// ---- FBs/Grid/FB_Grid_Power_Ext_Input.TcPOU
FUNCTION_BLOCK FB_Grid_Power_Ext_Input
VAR_INPUT PERSISTENT
	bEnable									: BOOL;													//Enable the Fuctionblock and his logic
	diNrOfEMS_IN							: DINT;													//Number of EMS on what this Device send Data
	rSizeGridConn							: REAL;													//{#lynus.ag#()} //Max Size of the Grid connection in kW
END_VAR
VAR_INPUT
	bExtErrorGrid							: BOOL;													//External Error for the Grid Function
	lrExtGridPower							: LREAL;												//External Grid power from a other Function or calculation in kW
	lrExtTotalCounterEnergy_Consumption		: LREAL;												//External Counter Value for Energy consumption with unit kWh
	lrExtTotalCounterEnergy_Production		: LREAL;												//External Counter Value for Energy production with unit kWh
	lrExtCounterEnergyT1_Consumption		: LREAL;												//External Counter Value for Energy consumption Tariff 1 with unit kWh
	lrExtCounterEnergyT2_Consumption		: LREAL;												//External Counter Value for Energy consumption Tariff 2 with unit kWh
	lrExtCounterEnergyT1_Production			: LREAL;												//External Counter Value for Energy production Tariff 1 with unit kWh
	lrExtCounterEnergyT2_Production			: LREAL;												//External Counter Value for Energy production Tariff 2 with unit kWh
END_VAR
VAR_OUTPUT
	stDataGrid								: ST_GridConnection_Output;								//{#lynus.ag#()} //Output Data from the Grid
	diNrOfGrid_OUT							: DINT;													//Active Number from the Grid connection for using on other functions
END_VAR
VAR
	{attribute 'hide'}
	fbGrid									: FB_GridConnection;									//Function block for grid connection
	{attribute 'hide'}
	fbNumberDevice							: FB_NumberOfDevice;									//Function block to calcualte the number of the Device
	{attribute 'hide'}
	timDissableFunctions					: TON;													//Timer to dissable the Function after Lynus_Standards.Constants_General.tTimeDissableLynusFunctions Days without connection to the Lynus Cloud
	{attribute 'hide'}
	timResetConnectionOnGVL					: TON;													//Timer to try reset the connection Flag on the GVL. (When somebody delete the Connection Function and make only a onlinechange)
	{attribute 'hide'}
	arrPD									: ARRAY[1..4] OF FB_PersistentData_Number;				//Function to save persistent data 
	{attribute 'hide'}
	byWaitInStep							: BYTE;													//Wait in Step before start to clean data on PLC
	{attribute 'hide'}
	iStateGVLData							: INT;													//State machine to handle the data on the GVL
	{attribute 'hide'}
	diCounterForGVL							: DINT;													//Counter to clean old data on GVL
	{attribute 'hide'}
	diLPForGVL								: DINT;													//Loop to clean old data on GVL
END_VAR
VAR PERSISTENT
	{attribute 'conditionalshow'}
	diNrOfEMS_IN_CP							: DINT;													//Number of EMS what control this Device to compare with the original
END_VAR

//Creator : Kai Ebensperger
//Company : Lynus AG
//Date : 07.06.2021
//Version : 1.0.0.0

//With this function block its possible to show the power data from a grid connection.
//The Power and Error Data came from a other Function and can connect to the Inputs. The Function write the Data then on the Lynus GVL
//The size from the Grid connection is sending to the ems

//NOTE for diNr.....Designation => 
//_IN = Here Data come in from other Functions or go out to other functions about the GVL
//_OUT = Here Data go out to other functions about the GVL

(*------------------------------------------------------------Limits----------------------------------------------------------------------------------*)

diNrOfEMS_IN := LIMIT(0,diNrOfEMS_IN,Constants_Energy.diMaxNumberOfEMS);

(*-------------------------------------------------------------Calcualte the number of Grid connection---------------------------------------------------------------*)

fbNumberDevice(
	diActualNumberOfDevices:= Lynus_Standards.GVL_Energy.stNumberOfDevices.diNumberOfGrids, 
	diMaxNumberOfDevices:= Constants_Energy.diMaxNumberOfGridConnections, 
	udiCounterOnlineChange:= TwinCAT_SystemInfoVarList._AppInfo.OnlineChangeCnt, 
	bNumberIsCalculatet=> , 
	bFPNumberIsCalculatet=> , 
	bOnlineChange=> , 
	diNumberForThisDevice=> diNrOfGrid_OUT, 
	diNumberOfTotalDevices=> );

//Write new Numer on GVL
IF fbNumberDevice.bFPNumberIsCalculatet THEN
	Lynus_Standards.GVL_Energy.stNumberOfDevices.diNumberOfGrids := fbNumberDevice.diNumberOfTotalDevices;	
END_IF 

//Delete old Number on GVL
IF fbNumberDevice.bOnlineChange THEN 
	Lynus_Standards.GVL_Energy.stNumberOfDevices.diNumberOfGrids := diNrOfGrid_OUT;	
		iStateGVLData := 1; 
END_IF	

(*-------------------------------------------------------------Service from Backend is ready and check the connection to backen for dissabel/enable Function---------------------------------------------------------------*)

//Try to reset the variable for connection on the GVL. When all is normal then the Lynus Mqtt connection function set this variable to true in the next cycle
//When we have no connection to the backend then after Lynus_Standards.Constants_General.tTimeDissableLynusFunctions days the Function is dissabled with all of his functionalities
timResetConnectionOnGVL(IN:= NOT timResetConnectionOnGVL.Q, PT:= T#1H, Q=> , ET=> );
	IF timResetConnectionOnGVL.Q THEN Lynus_Standards.GVL_Communicator.bStateConnectionToEnableFunctions := FALSE; END_IF
		IF NOT Lynus_Standards.GVL_Communicator.bStateConnectionToEnableFunctions THEN timDissableFunctions.IN := TRUE; ELSE timDissableFunctions.IN := FALSE; END_IF  
			timDissableFunctions(IN:= , PT:= Lynus_Standards.Constants_General.tTimeDissableLynusFunctions, Q=> , ET=> );

(*------------------------------------------------------------------Error----------------------------------------------------------------------------*)

IF timDissableFunctions.Q THEN fbGrid.bWarning := TRUE; fbGrid.iWarningCode := 0; ELSE fbGrid.bWarning := FALSE; END_IF 			
	IF bExtErrorGrid OR Lynus_Standards.GVL_Energy.stNumberOfDevices.diNumberOfGrids > Constants_Energy.diMaxNumberOfGridConnections THEN fbGrid.bError := TRUE; ELSE fbGrid.bError := FALSE; END_IF 

IF Lynus_Standards.GVL_Energy.stNumberOfDevices.diNumberOfGrids > Constants_Energy.diMaxNumberOfGridConnections THEN fbGrid.iErrorCode := 1;
ELSIF bExtErrorGrid THEN fbGrid.iErrorCode := 0;
END_IF  

(*------------------------------------------------------------------FB Grid----------------------------------------------------------------------------*)

fbGrid(
	bEnable:= bEnable AND NOT timDissableFunctions.Q, 
	bError:= , 
	bWriteWithDelay:= TRUE, 
	iErrorCode:= , 
	iWarningCode:= , 
	lrTotalCounterEnergy_Consumption:= lrExtTotalCounterEnergy_Consumption * 1000, 
	lrTotalCounterEnergy_Production:= lrExtTotalCounterEnergy_Production * 1000, 
	lrCounterEnergyT1_Consumption:= lrExtCounterEnergyT1_Consumption * 1000, 
	lrCounterEnergyT2_Consumption:= lrExtCounterEnergyT2_Consumption * 1000, 
	lrCounterEnergyT1_Production:= lrExtCounterEnergyT1_Production * 1000, 
	lrCounterEnergyT2_Production:= lrExtCounterEnergyT2_Production * 1000, 
	lrPowerGrid:= lrExtGridPower * 1000, 
	rSizeGridConn:= rSizeGridConn, 
	tTimDelayOutput:= T#5S, 
	stDataGridOut=> , 
	stDataGridOutDelay=> stDataGrid);
	
(*-----------------------------------------------------------Handle data to Global structure for the grid connections-----------------------------------------------------------------*)

//Delte al old Data on GVL after a online change or change on the variable diNrOfEMS_IDOD
IF diNrOfEMS_IN <> diNrOfEMS_IN_CP AND iStateGVLData = 0 THEN iStateGVLData := 10; END_IF 

CASE iStateGVLData OF
	
	0://Init Step
		byWaitInStep := 0;
			diCounterForGVL := 1;
	
	1://Wait for 4 Steps before clean al Data on GVL
		byWaitInStep := byWaitInStep + 1;
			IF byWaitInStep >= 4 AND fbNumberDevice.bNumberIsCalculatet THEN iStateGVLData := 2; END_IF
				//To much Devices, back to the Init step
				IF byWaitInStep >= 4 AND NOT fbNumberDevice.bNumberIsCalculatet THEN iStateGVLData := 0; END_IF	
			
	2://Clear all Data in GVL
		FOR diLPForGVL := 1 TO Constants_Energy.diMaxNumberOfEMS BY 1 DO 
			Lynus_Standards.GVL_Energy.stDataGridConnections[diLPForGVL,diCounterForGVL].bEnabled := FALSE;
				Lynus_Standards.GVL_Energy.stDataGridConnections[diLPForGVL,diCounterForGVL].byErrorWarning := 0;
					Lynus_Standards.GVL_Energy.stDataGridConnections[diLPForGVL,diCounterForGVL].lrPower := 0;
						Lynus_Standards.GVL_Energy.stDataGridConnections[diLPForGVL,diCounterForGVL].lrPowerConsumption := 0;
							Lynus_Standards.GVL_Energy.stDataGridConnections[diLPForGVL,diCounterForGVL].lrPowerProduction := 0;
								Lynus_Standards.GVL_Energy.stDataGridConnections[diLPForGVL,diCounterForGVL].rSizeGridConn := 0;
		END_FOR
			diCounterForGVL := diCounterForGVL + 1;
				diCounterForGVL := LIMIT(0,diCounterForGVL,Constants_Energy.diMaxNumberOfGridConnections);
					//Back to the init step
					IF diCounterForGVL >= Constants_Energy.diMaxNumberOfGridConnections THEN iStateGVLData := 0; END_IF

	10://Clear old Data on GVL 	
		Lynus_Standards.GVL_Energy.stDataGridConnections[diNrOfEMS_IN_CP,diNrOfGrid_OUT].bEnabled := FALSE;
			Lynus_Standards.GVL_Energy.stDataGridConnections[diNrOfEMS_IN_CP,diNrOfGrid_OUT].byErrorWarning := 0;
				Lynus_Standards.GVL_Energy.stDataGridConnections[diNrOfEMS_IN_CP,diNrOfGrid_OUT].lrPower := 0;
					Lynus_Standards.GVL_Energy.stDataGridConnections[diNrOfEMS_IN_CP,diNrOfGrid_OUT].lrPowerConsumption := 0;
						Lynus_Standards.GVL_Energy.stDataGridConnections[diNrOfEMS_IN_CP,diNrOfGrid_OUT].lrPowerProduction := 0;
							Lynus_Standards.GVL_Energy.stDataGridConnections[diNrOfEMS_IN_CP,diNrOfGrid_OUT].rSizeGridConn := 0;
	
		diNrOfEMS_IN_CP := diNrOfEMS_IN;
			//Back to the init step
			iStateGVLData := 0;

END_CASE 	 

IF diNrOfGrid_OUT > 0 AND fbNumberDevice.bNumberIsCalculatet AND diNrOfEMS_IN > 0 THEN
	Lynus_Standards.GVL_Energy.stDataGridConnections[diNrOfEMS_IN,diNrOfGrid_OUT].bEnabled := fbGrid.stDataGridOut.bEnabled;
		Lynus_Standards.GVL_Energy.stDataGridConnections[diNrOfEMS_IN,diNrOfGrid_OUT].byErrorWarning := fbGrid.stDataGridOut.byErrorWarning;
			Lynus_Standards.GVL_Energy.stDataGridConnections[diNrOfEMS_IN,diNrOfGrid_OUT].lrPower := fbGrid.stDataGridOut.lrPower;
				Lynus_Standards.GVL_Energy.stDataGridConnections[diNrOfEMS_IN,diNrOfGrid_OUT].lrPowerConsumption := fbGrid.stDataGridOut.lrPowerConsumption;
					Lynus_Standards.GVL_Energy.stDataGridConnections[diNrOfEMS_IN,diNrOfGrid_OUT].lrPowerProduction := fbGrid.stDataGridOut.lrPowerProduction;
						Lynus_Standards.GVL_Energy.stDataGridConnections[diNrOfEMS_IN,diNrOfGrid_OUT].rSizeGridConn := fbGrid.stDataGridOut.rSizeGridConn;
END_IF

(*----------------------------------------------------------Save persistent data----------------------------------------------------------------*)

arrPD[1](lrValue:= BOOL_TO_LREAL(bEnable), bEventBasedActive=> );
arrPD[2](lrValue:= DINT_TO_LREAL(diNrOfEMS_IN), bEventBasedActive=> );
arrPD[3](lrValue:= REAL_TO_LREAL(rSizeGridConn), bEventBasedActive=> );
arrPD[4](lrValue:= DINT_TO_LREAL(diNrOfEMS_IN_CP), bEventBasedActive=> );

END_FUNCTION_BLOCK

// ---- FBs/KBus State/FB_K_Bus_State_old.TcPOU
FUNCTION_BLOCK FB_K_Bus_State_old
VAR_INPUT
END_VAR
VAR_OUTPUT
	uiKBusState_OUT					AT%I*		: UINT;											//K-Bus State from the Basestation on wich the Terminal KL6301 is connected
END_VAR
VAR
END_VAR

//Creator : Kai Ebensperger
//Company : Lynus AG
//Date : 24.07.2021
//Version : 1.0.0.0

//With this Function Block its possible to connect the Variable on the output to the State Variable with the K-Bus Box
//In this Function we dont need code

END_FUNCTION_BLOCK

// ---- FBs/KBus State/FB_K_Bus_State.TcPOU
FUNCTION_BLOCK FB_K_Bus_State
VAR_INPUT
END_VAR
VAR_OUTPUT
	uiKBusState_OUT					AT%I*		: UINT;											//K-Bus State from the Basestation on wich the Terminal KL6301 is connected
	b_Kbus_notOk			: BOOL;			// KBus not OK, State <> 0
	word_ErrorCount			: WORD;			// Counts 1 up every time the KBus gets reset
END_VAR
VAR
	FB_IOF_DeviceReset	: IOF_DeviceReset;
    DEVICEID  : UDINT;
    RESET     : BOOL;
	ton_Delay_ResetKBus: Ton;
	Count_up: CTU;
END_VAR

//Creator : Stefan Lackner
//Company : EfficientIO
//Date : 09.02.2023
//Version : 1.0.0.0

//With this Function Block its possible to connect the Variable on the output to the State Variable with the K-Bus Box
//if the State <> 0 for longer then one Minute, the KBus gets reset

IF uiKBusState_OUT <> 0 AND NOT FB_IOF_DeviceReset.BUSY THEN
	ton_Delay_ResetKBus.IN := TRUE;
ELSE
	ton_Delay_ResetKBus.IN := FALSE;
END_IF
ton_Delay_ResetKBus( PT := T#1M);
 
FB_IOF_DeviceReset(
	NETID:= '', 
	DEVICEID:= 2, 		// ID 2 is the first terminal
	RESET:= ton_Delay_ResetKBus.Q, 
	TMOUT:= T#5S, 
	BUSY=> , 
	ERR=> , 
	ERRID=> );
	
IF uiKBusState_OUT <> 0 THEN
	b_Kbus_notOk := TRUE;
ELSE
	b_Kbus_notOk := FALSE;
END_IF

Count_up(
	CU:= b_Kbus_notOk, 
	RESET:= FALSE , 
	PV:= , 
	Q=> , 
	CV=> word_ErrorCount);

END_FUNCTION_BLOCK

// ---- FBs/MBus Master/FB_KL6781_MBus_Master.TcPOU
FUNCTION_BLOCK FB_KL6781_MBus_Master
VAR_INPUT PERSISTENT
	eBaudrateMBus							: E_MBus_Baudrate;				//With this Baudrate the Functionsblocks for the Counters are reading out
END_VAR
VAR_OUTPUT
	bBusy									: BOOL;							//Function is Busy
	bReady									: BOOL;							//Function is Ready
	byErrorWarning							: BYTE;							//Error Warning State
	diNrOfMBusMasterLine_OUT				: DINT;							//Active Number from the MBus Master Function for using on other functions
	eMessageMBusMaster						: E_Message_MBusMaster;			//Message from the MBus Master Function
END_VAR
VAR
	{attribute 'hide'}
	fbMbusMaster							: FB_MBUSKL6781;				//MBus Master for KL6781
	{attribute 'hide'}
	fbNumberDevice							: FB_NumberOfDevice;			//Function block to calcualte the number of the Device
	{attribute 'hide'}
	fbMBusMessage							: FB_MBusMaster_Messages;		//MBus Messages
	{attribute 'hide'}
	fbPD									: FB_PersistentData_Number;		//FB Persistent Data
	{attribute 'hide'}
	timDissableFunctions					: TON;							//Timer to dissable the Function after Lynus_Standards.Constants_General.tTimeDissableLynusFunctions Days without connection to the Lynus Cloud
	{attribute 'hide'}
	timResetConnectionOnGVL					: TON;							//Timer to try reset the connection Flag on the GVL. (When somebody delete the Connection Function and make only a onlinechange)
	stMBusKL6781ComIn        	AT%I*	 	: ST_KL6781inData22B;			//Input Structure for the KL6781 to map on the KL6781 Terminal
	stMBusKL6781ComOut        	AT%Q*		: ST_KL6781outData22B;			//Output Structure for the KL6781 to map on the KL6781 Terminal
	{attribute 'hide'}
	byWaitInStep							: BYTE;							//Wait in Step before start to clean data on PLC
	{attribute 'hide'}
	iStateGVLData							: INT;							//State machine to handle the data on the GVL
	{attribute 'hide'}
	diCounterForGVL							: DINT;							//Counter to clean old data on GVL
END_VAR

//Creator : Kai Ebensperger
//Company : Lynus AG
//Date : 23.07.2021
//Version : 1.0.0.0

//With this function block we can communicate with a beckhoff KL6781 MBus Terminal.
//This Functionblock receive the requests from the other Counter Functions and send to the Hardware Counters in the field.
//The answer from the Hardware Counters comes back to this Function and then they distribute to the Counter Function in the plc.
//This Function must be called in a task of < 10MS. Is depends about the Baudrate. 2400Baud = 10MS Task
//The request to a Hardware counter and the response is min. 1 second on MBus.


//NOTE for diNr.....Designation => 
//_IN = Here Data come in from other Functions or go out to other functions about the GVL
//_OUT = Here Data go out to other functions about the GVL

(*-------------------------------------------------------------Calcualte the number of MBus Master---------------------------------------------------------------*)

fbNumberDevice(
	diActualNumberOfDevices:= Lynus_Standards.GVL_Bussystems.diNumberOfMBusMasters, 
	diMaxNumberOfDevices:= Constants_Bussystems.diMaxNumberOfMBusMasterKL6781, 
	udiCounterOnlineChange:= TwinCAT_SystemInfoVarList._AppInfo.OnlineChangeCnt, 
	bNumberIsCalculatet=> , 
	bFPNumberIsCalculatet=> , 
	bOnlineChange=> , 
	diNumberForThisDevice=> diNrOfMBusMasterLine_OUT, 
	diNumberOfTotalDevices=> );

//Write new Numer on GVL
IF fbNumberDevice.bFPNumberIsCalculatet THEN
	Lynus_Standards.GVL_Bussystems.diNumberOfMBusMasters := fbNumberDevice.diNumberOfTotalDevices;	
END_IF 

//Delete old Number on GVL
IF fbNumberDevice.bOnlineChange THEN 
	Lynus_Standards.GVL_Bussystems.diNumberOfMBusMasters := diNrOfMBusMasterLine_OUT;	
		iStateGVLData := 1; 
END_IF	

(*-------------------------------------------------------------Service from Backend is ready and check the connection to backen for dissabel/enable Function---------------------------------------------------------------*)

//Try to reset the variable for connection on the GVL. When all is normal then the Lynus Mqtt connection function set this variable to true in the next cycle
//When we have no connection to the backend then after Lynus_Standards.Constants_General.tTimeDissableLynusFunctions days the Function is dissabled with all of his functionalities
timResetConnectionOnGVL(IN:= NOT timResetConnectionOnGVL.Q, PT:= T#1H, Q=> , ET=> );
	IF timResetConnectionOnGVL.Q THEN Lynus_Standards.GVL_Communicator.bStateConnectionToEnableFunctions := FALSE; END_IF
		IF NOT Lynus_Standards.GVL_Communicator.bStateConnectionToEnableFunctions THEN timDissableFunctions.IN := TRUE; ELSE timDissableFunctions.IN := FALSE; END_IF  
			timDissableFunctions(IN:= , PT:= Lynus_Standards.Constants_General.tTimeDissableLynusFunctions, Q=> , ET=> );
			
(*-------------------------------------------------------------M-Bus Master---------------------------------------------------------------*)

fbMbusMaster(
	usiRetries:= 0, 
	bStart:= , 
	bDisabled:= timDissableFunctions.Q OR diNrOfMBusMasterLine_OUT <= 0 OR NOT fbNumberDevice.bNumberIsCalculatet , 
	bBusy=> bBusy, 
	bReady=> bReady, 
	bError=> , 
	eError=> , 
	stComIn:= stMBusKL6781ComIn, 
	stComOut:= stMBusKL6781ComOut, 
	stCom:= Lynus_Standards.GVL_Bussystems.stDataOfMBusMasterKL6781[diNrOfMBusMasterLine_OUT].stDataMBusCommunicationKL6781);
	
(*------------------------------------------------------------------Error and Warning----------------------------------------------------------------------------*)
			
IF timDissableFunctions.Q THEN fbMBusMessage.bWarning := TRUE; fbMBusMessage.iWarningCode := 0; ELSE fbMBusMessage.bWarning := FALSE; END_IF   
	IF (Lynus_Standards.GVL_Bussystems.diNumberOfMBusMasters > Constants_Bussystems.diMaxNumberOfMBusMasterKL6781) THEN 
		fbMBusMessage.bErrorIntern := TRUE;
			fbMBusMessage.iErrorCode := 1;
	ELSE
		fbMBusMessage.bErrorIntern := FALSE;
	END_IF	

IF fbMbusMaster.bError THEN 
	fbMBusMessage.bErrorMBus := TRUE;
		fbMBusMessage.iErrorCode := fbMbusMaster.eError;
ELSE
	IF NOT fbMbusMaster.bError AND NOT fbMbusMaster.bBusy THEN 
		fbMBusMessage.bErrorMBus := FALSE;
	END_IF
END_IF	
		
fbMBusMessage(
	bErrorMBus:= , 
	bErrorIntern:= , 
	bWarning:= , 
	iWarningCode:= , 
	iErrorCode:= , 
	byErrorWarning=> byErrorWarning, 
	eMessageMBusMaster=> eMessageMBusMaster);
	
(*-----------------------------------------------------------Handle data to Global structure for MBus Communication-----------------------------------------------------------------*)
	
CASE iStateGVLData OF
	
	0://Init Step
		byWaitInStep := 0;
			diCounterForGVL := 1;
	
	1://Wait for 4 Steps before clean al Data on GVL
		byWaitInStep := byWaitInStep + 1;
			IF byWaitInStep >= 4 AND fbNumberDevice.bNumberIsCalculatet THEN iStateGVLData := 2; END_IF
				//To much Devices, back to the Init step
				IF byWaitInStep >= 4 AND NOT fbNumberDevice.bNumberIsCalculatet THEN iStateGVLData := 0; END_IF	
			
	2://Clear all Data in GVL
	//Some Parts in the GVL Reset the Slave. Otherwise there will be problems when writing the new addresses to the array in the GVL.
	
		Lynus_Standards.GVL_Bussystems.stDataOfMBusMasterKL6781[diCounterForGVL].eBaudrateMBusKL6781 := E_MBus_Baudrate.eMBus_NoBaudrate;
														 		
		diCounterForGVL := diCounterForGVL + 1;
			diCounterForGVL := LIMIT(0,diCounterForGVL,Constants_Bussystems.diMaxNumberOfMBusMasterKL6781);
				//Back to the init step
				IF diCounterForGVL >= Constants_Bussystems.diMaxNumberOfMBusMasterKL6781 THEN iStateGVLData := 0; END_IF

END_CASE 
	
IF diNrOfMBusMasterLine_OUT > 0 AND fbNumberDevice.bNumberIsCalculatet THEN  
	Lynus_Standards.GVL_Bussystems.stDataOfMBusMasterKL6781[diNrOfMBusMasterLine_OUT].eBaudrateMBusKL6781 := eBaudrateMBus;
END_IF	

(*----------------------------------------------------------Save persistent data----------------------------------------------------------------*)

fbPD(lrValue:= INT_TO_LREAL(eBaudrateMBus), bEventBasedActive=> );

END_FUNCTION_BLOCK

// ---- FBs/Meter/Beckhoff/Electric KL3403/FB_EM_Beckhoff_KL3403.TcPOU
FUNCTION_BLOCK FB_EM_Beckhoff_KL3403
VAR_INPUT PERSISTENT
	bEnable							: BOOL;											//Enable the function
	bChannel1Invers					: BOOL;											//Invert the Output data from Channel 1. = L1
	bChannel2Invers					: BOOL;											//Invert the Output data from Channel 2. = L2
	bChannel3Invers					: BOOL;											//Invert the Output data from Channel 3. = L3
	uiCurrentTransformerRatioL1		: UINT;											//Current Transformer Ratio for Channel 1 (L1)
	uiCurrentTransformerRatioL2		: UINT;											//Current Transformer Ratio for Channel 2 (L2)
	uiCurrentTransformerRatioL3		: UINT;											//Current Transformer Ratio for Channel 3 (L3)
END_VAR
VAR_INPUT
	uiKBusState_IN					: UINT;											//K-Bus State from the K-Bus Box on wich the Terminal is connected. (Connect with FB_K_Bus_state)
END_VAR
VAR_OUTPUT
	stDataEMPower					: ST_ElectricMeter_Output_Power;				//Output structure with Data from Electric Meter (Power Data)
	stDataEMCounter					: ST_ElectricMeter_Output_Counter;				//Output structure with Data from Electric Meter (Counter Data)
	stDataEMPowerRealTime			: ST_ElectricMeter_Output_Power;				//Output structure with Data from Electric Meter (Power Data RealTime)
	stDataEMCounterRealTime			: ST_ElectricMeter_Output_Counter;				//Output structure with Data from Electric Meter (Counter Data RealTime)
	diNrOfEM_OUT					: DINT;											//Active Number from the Electric Meter for using on other functions
END_VAR
VAR
	{attribute 'conditionalshow'}
	fbEM							: FB_ElectricMeter;								//Electric Meter Function
	{attribute 'conditionalshow'}
	fbEnergyCounter					: FB_EnergyCounter;								//FB energy Counter, because the KL3403 has no nice logic for the Energy value
	{attribute 'hide'}
	fbNumberDevice					: FB_NumberOfDevice;							//Function block to calcualte the number of the Device
	fbKL3403						: FB_KL3403_SimpleProcessImage;					//Function KL3403
	{attribute 'hide'}
	stDataL1						: ST_KL3403;									//Data from Channel 1 (L1)
	{attribute 'hide'}
	stDataL2						: ST_KL3403;									//Data from Channel 2 (L2)
	{attribute 'hide'}
	stDataL3						: ST_KL3403;									//Data from Channel 3 (L3)
	{attribute 'hide'}
	timDissableFunctions			: TON;											//Timer to dissable the Function after Lynus_Standards.Constants_General.tTimeDissableLynusFunctions Days without connection to the Lynus Cloud
	{attribute 'hide'}
	timResetConnectionOnGVL			: TON;											//Timer to try reset the connection Flag on the GVL. (When somebody delete the Connection Function and make only a onlinechange)
	{attribute 'hide'}
	timSetCounterValues				: TON;											//Timer to set the counter values from the KL3403 Function to the EM Function
	{attribute 'hide'}
	arrPD							: ARRAY[1..7] OF FB_PersistentData_Number;		//Function to save persistent data
	{attribute 'hide'}
	byWaitInStep					: BYTE;											//Wait in Step before start to clean data on PLC
	{attribute 'hide'}
	iStateGVLData					: INT;											//State machine to handle the data on the GVL
	{attribute 'hide'}
	diCounterForGVL					: DINT;											//Counter to clean old data on GVL
END_VAR

//Creator : Kai Ebensperger
//Company : Lynus AG
//Date : 04.10.2021
//Version : 1.0.0.0

//Stefan: Addes S and Q calculation

//With this function is possible to read out all Information from a KL3403
//This Function support only the Simple Process Image and the Ratio in the Terminal register must be Set allways to 1.

//NOTE for diNr.....Designation => 
//_IN = Here Data come in from other Functions or go out to other functions about the GVL
//_OUT = Here Data go out to other functions about the GVL

(*-------------------------------------------------------------Calcualte the number of EM---------------------------------------------------------------*)

fbNumberDevice(
	diActualNumberOfDevices:= Lynus_Standards.GVL_Energy.stNumberOfDevices.diNumberOfElectricMeters, 
	diMaxNumberOfDevices:= Constants_Energy.diMaxNumberOfElectricMeters, 
	udiCounterOnlineChange:= TwinCAT_SystemInfoVarList._AppInfo.OnlineChangeCnt, 
	bNumberIsCalculatet=> , 
	bFPNumberIsCalculatet=> , 
	bOnlineChange=> , 
	diNumberForThisDevice=> diNrOfEM_OUT, 
	diNumberOfTotalDevices=> );

//Write new Numer on GVL
IF fbNumberDevice.bFPNumberIsCalculatet THEN
	Lynus_Standards.GVL_Energy.stNumberOfDevices.diNumberOfElectricMeters := fbNumberDevice.diNumberOfTotalDevices;	
END_IF

//Delete old Number on GVL
IF fbNumberDevice.bOnlineChange THEN 
	Lynus_Standards.GVL_Energy.stNumberOfDevices.diNumberOfElectricMeters := diNrOfEM_OUT;	
		iStateGVLData := 1; 
END_IF

(*-------------------------------------------------------------Service from Backend is ready and check the connection to backen for dissabel/enable Function---------------------------------------------------------------*)

//Try to reset the variable for connection on the GVL. When all is normal then the Lynus Mqtt connection function set this variable to true in the next cycle
//When we have no connection to the backend then after Lynus_Standards.Constants_General.tTimeDissableLynusFunctions days the Function is dissabled with all of his functionalities
timResetConnectionOnGVL(IN:= NOT timResetConnectionOnGVL.Q, PT:= T#1H, Q=> , ET=> );
	IF timResetConnectionOnGVL.Q THEN Lynus_Standards.GVL_Communicator.bStateConnectionToEnableFunctions := FALSE; END_IF
		IF NOT Lynus_Standards.GVL_Communicator.bStateConnectionToEnableFunctions THEN timDissableFunctions.IN := TRUE; ELSE timDissableFunctions.IN := FALSE; END_IF  
			timDissableFunctions(IN:= , PT:= Lynus_Standards.Constants_General.tTimeDissableLynusFunctions, Q=> , ET=> );

(*----------------------------------------------------------------------------------------KL3403 Communication----------------------------------------------------------------------------------------------*)

fbKL3403(
	uiKBusState_IN:= uiKBusState_IN, 
	uiCurrentTransformerRatioL1:= uiCurrentTransformerRatioL1,
	uiCurrentTransformerRatioL2:= uiCurrentTransformerRatioL2,
	uiCurrentTransformerRatioL3:= uiCurrentTransformerRatioL3,
	rResolutionCurrent:= 0.001,
	rResolutionPower:= 0.1,
	rResolutionEnergy:= 0.01,
	stDataL1=> , 
	stDataL2=> ,
	stDataL3=> );

//Invert the Output data, because it is possible that the current transformers have been mounted in different mounting positions.
IF NOT bChannel1Invers THEN
	stDataL1 := fbKL3403.stDataL1;
ELSE
	stDataL1.byErrorWarning := fbKL3403.stDataL1.byErrorWarning;
	stDataL1.rCurrent := fbKL3403.stDataL1.rCurrent;
	stDataL1.rVoltage := fbKL3403.stDataL1.rVoltage;
	stDataL1.rPower := fbKL3403.stDataL1.rPower * - 1;
	stDataL1.rPowerfactor := fbKL3403.stDataL1.rPowerfactor;
	stDataL1.rEnergy := fbKL3403.stDataL1.rEnergy;
	stDataL1.rFrequency := fbKL3403.stDataL1.rFrequency;
	stDataL1.rPeakValueCurrent := fbKL3403.stDataL1.rPeakValueCurrent;
	stDataL1.rPeakValueVoltage := fbKL3403.stDataL1.rPeakValueVoltage;
	stDataL1.rPeakValuePower := fbKL3403.stDataL1.rPeakValuePower * - 1;
	stDataL1.rMinValueCurrent := fbKL3403.stDataL1.rMinValueCurrent;
	stDataL1.rMinValueVoltage := fbKL3403.stDataL1.rMinValueVoltage;
	stDataL1.rMinValuePower := fbKL3403.stDataL1.rMinValuePower * - 1;
END_IF

IF NOT bChannel2Invers THEN
	stDataL2 := fbKL3403.stDataL2;
ELSE
	stDataL2.byErrorWarning := fbKL3403.stDataL2.byErrorWarning;
	stDataL2.rCurrent := fbKL3403.stDataL2.rCurrent;
	stDataL2.rVoltage := fbKL3403.stDataL2.rVoltage;
	stDataL2.rPower := fbKL3403.stDataL2.rPower * - 1;
	stDataL2.rPowerfactor := fbKL3403.stDataL2.rPowerfactor;
	stDataL2.rEnergy := fbKL3403.stDataL2.rEnergy;
	stDataL2.rFrequency := fbKL3403.stDataL2.rFrequency;
	stDataL2.rPeakValueCurrent := fbKL3403.stDataL2.rPeakValueCurrent;
	stDataL2.rPeakValueVoltage := fbKL3403.stDataL2.rPeakValueVoltage;
	stDataL2.rPeakValuePower := fbKL3403.stDataL2.rPeakValuePower * - 1;
	stDataL2.rMinValueCurrent := fbKL3403.stDataL2.rMinValueCurrent;
	stDataL2.rMinValueVoltage := fbKL3403.stDataL2.rMinValueVoltage;
	stDataL2.rMinValuePower := fbKL3403.stDataL2.rMinValuePower * - 1;
END_IF

IF NOT bChannel3Invers THEN
	stDataL3 := fbKL3403.stDataL3;
ELSE
	stDataL3.byErrorWarning := fbKL3403.stDataL3.byErrorWarning;
	stDataL3.rCurrent := fbKL3403.stDataL3.rCurrent;
	stDataL3.rVoltage := fbKL3403.stDataL3.rVoltage;
	stDataL3.rPower := fbKL3403.stDataL3.rPower * - 1;
	stDataL3.rPowerfactor := fbKL3403.stDataL3.rPowerfactor;
	stDataL3.rEnergy := fbKL3403.stDataL3.rEnergy;
	stDataL3.rFrequency := fbKL3403.stDataL3.rFrequency;
	stDataL3.rPeakValueCurrent := fbKL3403.stDataL3.rPeakValueCurrent;
	stDataL3.rPeakValueVoltage := fbKL3403.stDataL3.rPeakValueVoltage;
	stDataL3.rPeakValuePower := fbKL3403.stDataL3.rPeakValuePower * - 1;
	stDataL3.rMinValueCurrent := fbKL3403.stDataL3.rMinValueCurrent;
	stDataL3.rMinValueVoltage := fbKL3403.stDataL3.rMinValueVoltage;
	stDataL3.rMinValuePower := fbKL3403.stDataL3.rMinValuePower * - 1;
END_IF
	
(*----------------------------------------------------------------------------------------Energy Counter Function----------------------------------------------------------------------------------------------*)

//For the KL3403 we use a external Energy Counter Function. So we can count Import and Export Energy with the KL3403.
//Attetntion, the KL3403 is not MID Conform. Thus, these values must not be used for billing.
fbEnergyCounter(
	byActiveTariff:= 1, 
	lrPowerInput:= (stDataL1.rPower + stDataL2.rPower + stDataL3.rPower) / 1000, 
	lrTotalCounterEnergy_Consumption=> , 
	lrTotalCounterEnergy_Production=> , 
	lrCounterEnergyT1_Consumption=> , 
	lrCounterEnergyT2_Consumption=> , 
	lrCounterEnergyT1_Production=> , 
	lrCounterEnergyT2_Production=> );

(*----------------------------------------------------------------------------------------Electric Meter Function----------------------------------------------------------------------------------------------*)

//Error
IF timDissableFunctions.Q THEN fbEM.bWarning := TRUE; fbEM.iWarningCode := 0; ELSE fbEM.bWarning := FALSE; END_IF 
	IF Lynus_Standards.GVL_Energy.stNumberOfDevices.diNumberOfElectricMeters > Constants_Energy.diMaxNumberOfElectricMeters OR 
		stDataL1.byErrorWarning = 2 OR stDataL2.byErrorWarning = 2 OR stDataL3.byErrorWarning = 2 THEN 
			fbEM.bError := TRUE; 
	ELSE 
			fbEM.bError := FALSE; 
	END_IF
		IF Lynus_Standards.GVL_Energy.stNumberOfDevices.diNumberOfElectricMeters > Constants_Energy.diMaxNumberOfElectricMeters THEN fbEM.iErrorCode := 1;
		ELSIF stDataL1.byErrorWarning = 2 OR stDataL2.byErrorWarning = 2 OR stDataL3.byErrorWarning = 2 THEN fbEM.iErrorCode := 0;
		END_IF

timSetCounterValues(IN:= bEnable AND NOT timSetCounterValues.Q, PT:= T#2S, Q=> , ET=> );		

//Function
fbEM(
	bEnable:= bEnable AND NOT timDissableFunctions.Q, 
	bError:= , 
	bEnableReadOutFunction:= FALSE, 
	bWriteWithDelay:= TRUE, 
	bPowerDataInvers:= FALSE,
	bReadOutDataDone:= timSetCounterValues.Q,
	iTimeReadOutInterval:= 0, 
	iErrorCode:= , 
	iWarningCode:= , 
	lrTotalCounterEnergy_Consumption:= fbEnergyCounter.lrTotalCounterEnergy_Consumption,
	lrTotalCounterEnergy_Production:= fbEnergyCounter.lrTotalCounterEnergy_Production, 
	lrCounterEnergyT1_Consumption:= fbEnergyCounter.lrCounterEnergyT1_Consumption,
	lrCounterEnergyT2_Consumption:= fbEnergyCounter.lrCounterEnergyT2_Consumption,
	lrCounterEnergyT1_Production:= fbEnergyCounter.lrCounterEnergyT1_Production, 
	lrCounterEnergyT2_Production:= fbEnergyCounter.lrCounterEnergyT2_Production, 
	lrCurrentL1:= stDataL1.rCurrent, 
	lrVoltageL1N:= stDataL1.rVoltage, 
	lrVoltageL1L2:= stDataL1.rVoltage*SQRT(3), 
	lrPowerL1:= stDataL1.rPower, 
	lrCurrentL2:= stDataL2.rCurrent, 
	lrVoltageL2N:= stDataL2.rVoltage, 
	lrVoltageL2L3:= stDataL2.rVoltage*SQRT(3), 
	lrPowerL2:= stDataL2.rPower, 
	lrCurrentL3:= stDataL3.rCurrent, 
	lrVoltageL3N:= stDataL3.rVoltage, 
	lrVoltageL3L1:= stDataL3.rVoltage*SQRT(3), 
	lrPowerL3:= stDataL3.rPower, 
	lrPowerTotal:= stDataL1.rPower + stDataL2.rPower + stDataL3.rPower, 
	lrFrequency:= (stDataL1.rFrequency + stDataL2.rFrequency + stDataL3.rFrequency) / 3, 
 	lrApparentPowerTotal:=,
	lrReactivePowerTotal:=, 
	tTimDelayOutput:= T#5S, 
	stDataEMOutPower=> stDataEMPowerRealTime, 
	stDataEMOutPowerDelay=> stDataEMPower, 
	stDataEMOutCounter=> stDataEMCounterRealTime,
	stDataEMOutCounterDelay=> stDataEMCounter,
	bReadOutMeter=> );
(*
	IF  stDataL1.rPowerfactor <>0 AND stDataL2.rPowerfactor <>0 AND stDataL3.rPowerfactor <>0 THEN
		fbEM.lrApparentPowerTotal:= ABS(stDataL1.rPower)/ABS(stDataL1.rPowerfactor) + ABS(stDataL2.rPower)/ABS(stDataL2.rPowerfactor) + ABS(stDataL3.rPower)/ABS(stDataL3.rPowerfactor); 
	END_IF	
*)


	//calculate total apparant power in VA
	fbEM.lrApparentPowerTotal := fbEM.lrVoltageL1N * fbEM.lrCurrentL1 + fbEM.lrVoltageL2N * fbEM.lrCurrentL2 +  fbEM.lrVoltageL3N * fbEM.lrCurrentL3;
	
	IF fbEM.lrApparentPowerTotal<>0 AND fbEM.lrPowerTotal<>0 AND fbEM.lrApparentPowerTotal> ABS(fbEM.lrPowerTotal) THEN
		fbEM.lrReactivePowerTotal:= SQRT(ABS(fbEM.lrApparentPowerTotal*fbEM.lrApparentPowerTotal - ABS(fbEM.lrPowerTotal*fbEM.lrPowerTotal)));	
	END_IF
	IF stDataL1.rPowerfactor<>0 AND stDataL2.rPowerfactor <>0 AND stDataL3.rPowerfactor<>0 THEN 	// check that not all cos phi are not 0
		IF (stDataL1.rPowerfactor+stDataL2.rPowerfactor+stDataL3.rPowerfactor)<>0 THEN				// check that the sum is not 0	
			IF 	(stDataL1.rPowerfactor+stDataL2.rPowerfactor+stDataL3.rPowerfactor)/3<0 THEN		// check is the average is below 0 / capacitive
				fbEM.lrReactivePowerTotal:=fbEM.lrReactivePowerTotal*(-1);
			END_IF
		END_IF	
	END_IF
(*-----------------------------------------------------------Handle data to Global structure for Electric Meter-----------------------------------------------------------------*)

CASE iStateGVLData OF
	
	0://Init Step
		byWaitInStep := 0;
			diCounterForGVL := 1;
	
	1://Wait for 4 Steps before clean al Data on GVL
		byWaitInStep := byWaitInStep + 1;
			IF byWaitInStep >= 4 AND fbNumberDevice.bNumberIsCalculatet THEN iStateGVLData := 2; END_IF
				//To much Devices, back to the Init step
				IF byWaitInStep >= 4 AND NOT fbNumberDevice.bNumberIsCalculatet THEN iStateGVLData := 0; END_IF	
			
	2://Clear all Data in GVL
		Lynus_Standards.GVL_Energy.stDataElectricMeters[diCounterForGVL].bEnabled := FALSE;	
			Lynus_Standards.GVL_Energy.stDataElectricMeters[diCounterForGVL].byErrorWarning := 0;
				Lynus_Standards.GVL_Energy.stDataElectricMeters[diCounterForGVL].lrCounterEnergyT1_Consumption := 0;
					Lynus_Standards.GVL_Energy.stDataElectricMeters[diCounterForGVL].lrCounterEnergyT1_Production := 0;
						Lynus_Standards.GVL_Energy.stDataElectricMeters[diCounterForGVL].lrCounterEnergyT2_Consumption := 0;
							Lynus_Standards.GVL_Energy.stDataElectricMeters[diCounterForGVL].lrCounterEnergyT2_Production := 0;
								Lynus_Standards.GVL_Energy.stDataElectricMeters[diCounterForGVL].lrPower := 0;
									Lynus_Standards.GVL_Energy.stDataElectricMeters[diCounterForGVL].lrPowerConsumption := 0;
										Lynus_Standards.GVL_Energy.stDataElectricMeters[diCounterForGVL].lrPowerProduction := 0;
											Lynus_Standards.GVL_Energy.stDataElectricMeters[diCounterForGVL].lrTotalCounterEnergy_Consumption := 0;
												Lynus_Standards.GVL_Energy.stDataElectricMeters[diCounterForGVL].lrTotalCounterEnergy_Production := 0;
		
		//Electric Meters
		diCounterForGVL := diCounterForGVL + 1;
			diCounterForGVL := LIMIT(0,diCounterForGVL,Constants_Energy.diMaxNumberOfElectricMeters);
				//Back to the init step
				IF diCounterForGVL >= Constants_Energy.diMaxNumberOfElectricMeters THEN iStateGVLData := 0; END_IF

END_CASE 	 

//Write Data on GVL for Electric Meter
IF diNrOfEM_OUT > 0 AND fbNumberDevice.bNumberIsCalculatet THEN
	Lynus_Standards.GVL_Energy.stDataElectricMeters[diNrOfEM_OUT].bEnabled := fbEM.stDataEMOutPower.bEnabled;
		Lynus_Standards.GVL_Energy.stDataElectricMeters[diNrOfEM_OUT].byErrorWarning := fbEM.stDataEMOutPower.byErrorWarning;
			Lynus_Standards.GVL_Energy.stDataElectricMeters[diNrOfEM_OUT].lrCounterEnergyT1_Consumption := fbEM.stDataEMOutCounter.lrCounterEnergyT1_Consumption;
				Lynus_Standards.GVL_Energy.stDataElectricMeters[diNrOfEM_OUT].lrCounterEnergyT1_Production := fbEM.stDataEMOutCounter.lrCounterEnergyT1_Production;
					Lynus_Standards.GVL_Energy.stDataElectricMeters[diNrOfEM_OUT].lrCounterEnergyT2_Consumption := fbEM.stDataEMOutCounter.lrCounterEnergyT2_Consumption;
						Lynus_Standards.GVL_Energy.stDataElectricMeters[diNrOfEM_OUT].lrCounterEnergyT2_Production := fbEM.stDataEMOutCounter.lrCounterEnergyT2_Production;		
							Lynus_Standards.GVL_Energy.stDataElectricMeters[diNrOfEM_OUT].lrPower := fbEM.stDataEMOutPower.lrPowerTotal;
								Lynus_Standards.GVL_Energy.stDataElectricMeters[diNrOfEM_OUT].lrPowerConsumption := fbEM.stDataEMOutPower.lrPowerConsumption;
									Lynus_Standards.GVL_Energy.stDataElectricMeters[diNrOfEM_OUT].lrPowerProduction := fbEM.stDataEMOutPower.lrPowerProduction;
										Lynus_Standards.GVL_Energy.stDataElectricMeters[diNrOfEM_OUT].lrTotalCounterEnergy_Consumption := fbEM.stDataEMOutCounter.lrTotalCounterEnergy_Consumption;
											Lynus_Standards.GVL_Energy.stDataElectricMeters[diNrOfEM_OUT].lrTotalCounterEnergy_Production := fbEM.stDataEMOutCounter.lrTotalCounterEnergy_Production;
END_IF

(*----------------------------------------------------------Save persistent data----------------------------------------------------------------*)

arrPD[1](lrValue:= BOOL_TO_LREAL(bEnable), bEventBasedActive=> );
arrPD[2](lrValue:= UINT_TO_LREAL(uiCurrentTransformerRatioL1), bEventBasedActive=> );
arrPD[3](lrValue:= UINT_TO_LREAL(uiCurrentTransformerRatioL2), bEventBasedActive=> );
arrPD[4](lrValue:= UINT_TO_LREAL(uiCurrentTransformerRatioL3), bEventBasedActive=> );
arrPD[5](lrValue:= BOOL_TO_LREAL(bChannel1Invers), bEventBasedActive=> );
arrPD[6](lrValue:= BOOL_TO_LREAL(bChannel2Invers), bEventBasedActive=> );
arrPD[7](lrValue:= BOOL_TO_LREAL(bChannel3Invers), bEventBasedActive=> );

END_FUNCTION_BLOCK

// ---- FBs/Electric Charging Station/Linear AO/FB_ECS_Linear_AO.TcPOU
FUNCTION_BLOCK FB_ECS_Linear_AO
VAR_INPUT PERSISTENT
	bEnable									: BOOL;											//{#lynus.ag#()} //Enable the Fuctionblock and his logic
	bPowerDataInvers						: BOOL;											//With True its possible to invert all received power data from the electric meter
	bNoLinear								: BOOL;											//Output Power from the device is not linear. Use the Values from the Table Of Interpolation Points.
	byElectricFuseLine						: BYTE; 										//Electric Fuse Line on wich the ECS is connected => 1 2 3 (If 0 then this charging station is not connected to a Electric Fuse Line)
	diNrOfEMS_IN							: DINT;											//Number of EMS what control this Device.
	diNrOfEM_IN_CS							: DINT;											//Number of the electric meter for incoming power data. (Power Data for this Device)
	stSetupECS								: ST_Setup_ECS;									//{#lynus.ag#()} //Setup charging station
	arrTableOfInterpolationPoints			: ARRAY[1..10] OF REAL;							//Table Of Interpolation Points. Corresponds to the different power values in the non-linear curve of the device. The last value must correspond to the maximum power.
END_VAR
VAR_INPUT
	bCarConnectedExt						: BOOL;											//Car connected signal from external function			
	bErrorExt								: BOOL;											//Error Signal from external Function
	bWarningExt								: BOOL;											//Warning Signal from external Function 						
END_VAR
VAR_OUTPUT
	stDataECS								: ST_ECS_Output;								//{#lynus.ag#()} //Electric charging station output data
	diNrOfECS_OUT							: DINT;											//Active Number from the Electric charging Function for using on other functions
	rTargetPowerForExtFunc					: REAL;											//Target Power from 0% to +100% to use on a external Function
	rTargetChargCurrentForExtFunc			: REAL;											//Target charge Current to use on a external Function
END_VAR
VAR
	{attribute 'hide'}
	fbCS									: FB_ElectricChargingStation;					//Function block for electric charging station
	{attribute 'hide'}
	fbNumberDevice							: FB_NumberOfDevice;							//Function block to calcualte the number of the Device
	{attribute 'hide'}
	fbInterpolation							: FB_Lin_Interpolation;							//Function for interpolation
	fbDIExternalLock						: FB_XL1XXX_DI;									//Digital Input from external loock signal
	fbAOCS									: FB_XL4XXX_AO;									//Analog Output to swtich on and off the charging station
	{attribute 'hide'}
	timDissableFunctions					: TON;											//Timer to dissable the Function after Lynus_Standards.Constants_General.tTimeDissableLynusFunctions Days without connection to the Lynus Cloud
	{attribute 'hide'}
	timResetConnectionOnGVL					: TON;											//Timer to try reset the connection Flag on the GVL. (When somebody delete the Connection Function and make only a onlinechange)
	{attribute 'hide'}
	arrPD									: ARRAY[1..25] OF FB_PersistentData_Number;		//Function to save persistent data 
	{attribute 'hide'}
	byWaitInStep							: BYTE;											//Wait in Step before start to clean data on PLC
	{attribute 'hide'}
	iStateGVLData							: INT;											//State machine to handle the data on the GVL
	{attribute 'hide'}
	diNumberOfActiveBatterys				: DINT;											//Number of active batterys
	{attribute 'hide'}
	diNumberOfBatteryInverterInEPO			: DINT;											//Number of battery inverters that work in Emergency Power operation 
	{attribute 'hide'}
	diCounterForGVL							: DINT;											//Counter to clean old data on GVL
	{attribute 'hide'}
	diLPForGVL								: DINT;											//Loop to clean old data on GVL
	{attribute 'hide'}
	dwSumSOC								: DWORD;										//Sum of the SOC from all batterys	
	{attribute 'hide'}
	liLPBatteryData							: LINT;											//Loop to check some data from batterys
	{attribute 'hide'}
	liLPInEPO								: LINT;											//Loop to check if 1 or more battery inverters build a island grid
END_VAR
VAR PERSISTENT
	{attribute 'conditionalshow'}
	diNrOfEMS_IN_CP							: DINT;											//Number of EMS what control this Device to compare with the original
END_VAR

//Creator : Kai Ebensperger
//Company : Lynus AG
//Date : 19.05.2021
//Version : 1.0.0.0

//With this function block its possible to switch on and off a charging station
//Its also possible to control the target power with the analog output signal
//With the Nr from the Electric Meter its possible to send the data fromt the electric meter directly to the CS function to display it

//NOTE for diNr.....Designation => 
//_IN = Here Data come in from other Functions or go out to other functions about the GVL
//_OUT = Here Data go out to other functions about the GVL

(*------------------------------------------------------------Limits----------------------------------------------------------------------------------*)

diNrOfEMS_IN := LIMIT(0,diNrOfEMS_IN,Constants_Energy.diMaxNumberOfEMS);
	diNrOfEM_IN_CS := LIMIT(0,diNrOfEM_IN_CS,Constants_Energy.diMaxNumberOfElectricMeters);	
		byElectricFuseLine := LIMIT(0,byElectricFuseLine,30);	
			
(*------------------------------------------------------------------Power Data----------------------------------------------------------------------------*)

//Energy Session Input data
fbCS.bCalculateEnergySession := FALSE;
fbCS.arrSocketPowerECS[1] := 0;
fbCS.arrSocketPowerECS[2] := 0;
fbCS.arrSocketPowerECS[3] := 0;
fbCS.arrSocketPowerECS[4] := 0;
fbCS.arrSocketEnergySession[1] := 0;
fbCS.arrSocketEnergySession[2] := 0;
fbCS.arrSocketEnergySession[3] := 0;
fbCS.arrSocketEnergySession[4] := 0;

IF NOT bPowerDataInvers THEN
	fbCS.lrCounterEnergyT1_Consumption := Lynus_Standards.GVL_Energy.stDataElectricMeters[diNrOfEM_IN_CS].lrCounterEnergyT1_Production * 1000;
	fbCS.lrCounterEnergyT2_Consumption := Lynus_Standards.GVL_Energy.stDataElectricMeters[diNrOfEM_IN_CS].lrCounterEnergyT2_Production * 1000;
	fbCS.lrCounterEnergyT1_Production := Lynus_Standards.GVL_Energy.stDataElectricMeters[diNrOfEM_IN_CS].lrCounterEnergyT1_Consumption * 1000;
	fbCS.lrCounterEnergyT2_Production := Lynus_Standards.GVL_Energy.stDataElectricMeters[diNrOfEM_IN_CS].lrCounterEnergyT1_Consumption * 1000;
	fbCS.lrTotalCounterEnergy_Consumption := Lynus_Standards.GVL_Energy.stDataElectricMeters[diNrOfEM_IN_CS].lrTotalCounterEnergy_Production * 1000;
	fbCS.lrTotalCounterEnergy_Production := Lynus_Standards.GVL_Energy.stDataElectricMeters[diNrOfEM_IN_CS].lrTotalCounterEnergy_Consumption * 1000;
		fbCS.lrTotalPowerECS := (Lynus_Standards.GVL_Energy.stDataElectricMeters[diNrOfEM_IN_CS].lrPower * 1000) * - 1;
ELSE
	fbCS.lrCounterEnergyT1_Consumption := Lynus_Standards.GVL_Energy.stDataElectricMeters[diNrOfEM_IN_CS].lrCounterEnergyT1_Consumption * 1000;
	fbCS.lrCounterEnergyT2_Consumption := Lynus_Standards.GVL_Energy.stDataElectricMeters[diNrOfEM_IN_CS].lrCounterEnergyT2_Consumption * 1000;
	fbCS.lrCounterEnergyT1_Production := Lynus_Standards.GVL_Energy.stDataElectricMeters[diNrOfEM_IN_CS].lrCounterEnergyT1_Production * 1000;
	fbCS.lrCounterEnergyT2_Production := Lynus_Standards.GVL_Energy.stDataElectricMeters[diNrOfEM_IN_CS].lrCounterEnergyT2_Production * 1000;
	fbCS.lrTotalCounterEnergy_Consumption := Lynus_Standards.GVL_Energy.stDataElectricMeters[diNrOfEM_IN_CS].lrTotalCounterEnergy_Consumption * 1000;
	fbCS.lrTotalCounterEnergy_Production := Lynus_Standards.GVL_Energy.stDataElectricMeters[diNrOfEM_IN_CS].lrTotalCounterEnergy_Production * 1000;
		fbCS.lrTotalPowerECS := Lynus_Standards.GVL_Energy.stDataElectricMeters[diNrOfEM_IN_CS].lrPower * 1000;
END_IF

(*-------------------------------------------------------------Calcualte the number of ECS---------------------------------------------------------------*)

fbNumberDevice(
	diActualNumberOfDevices:= Lynus_Standards.GVL_Energy.stNumberOfDevices.diNumberOfECS, 
	diMaxNumberOfDevices:= Constants_Energy.diMaxNumberOfElectricChargingStations, 
	udiCounterOnlineChange:= TwinCAT_SystemInfoVarList._AppInfo.OnlineChangeCnt, 
	bNumberIsCalculatet=> , 
	bFPNumberIsCalculatet=> , 
	bOnlineChange=> , 
	diNumberForThisDevice=> diNrOfECS_OUT, 
	diNumberOfTotalDevices=> );

//Write new Numer on GVL
IF fbNumberDevice.bFPNumberIsCalculatet THEN
	Lynus_Standards.GVL_Energy.stNumberOfDevices.diNumberOfECS := fbNumberDevice.diNumberOfTotalDevices;	
END_IF 

//Delete old Number on GVL
IF fbNumberDevice.bOnlineChange THEN 
	Lynus_Standards.GVL_Energy.stNumberOfDevices.diNumberOfECS := diNrOfECS_OUT;	
		iStateGVLData := 1; 
END_IF

(*-------------------------------------------------------------Service from Backend is ready and check the connection to backend for dissabel/enable Function---------------------------------------------------------------*)

//Try to reset the variable for connection on the GVL. When all is normal then the Lynus Mqtt connection function set this variable to true in the next cycle
//When we have no connection to the backend then after Lynus_Standards.Constants_General.tTimeDissableLynusFunctions days the Function is dissabled with all of his functionalities
timResetConnectionOnGVL(IN:= NOT timResetConnectionOnGVL.Q, PT:= T#1H, Q=> , ET=> );
	IF timResetConnectionOnGVL.Q THEN Lynus_Standards.GVL_Communicator.bStateConnectionToEnableFunctions := FALSE; END_IF
		IF NOT Lynus_Standards.GVL_Communicator.bStateConnectionToEnableFunctions THEN timDissableFunctions.IN := TRUE; ELSE timDissableFunctions.IN := FALSE; END_IF  
			timDissableFunctions(IN:= , PT:= Lynus_Standards.Constants_General.tTimeDissableLynusFunctions, Q=> , ET=> );	

(*------------------------------------------------------------------Error and Warning----------------------------------------------------------------------------*)	

IF timDissableFunctions.Q OR bWarningExt THEN fbCS.bWarning := TRUE; ELSE fbCS.bWarning := FALSE; END_IF   
	IF Lynus_Standards.GVL_Energy.stNumberOfDevices.diNumberOfECS > Constants_Energy.diMaxNumberOfElectricChargingStations OR bErrorExt THEN 
		fbCS.bError := TRUE;
	ELSE 
		fbCS.bError := FALSE;
	END_IF

IF timDissableFunctions.Q THEN fbCS.iWarningCode := 0;
ELSIF bWarningExt THEN fbCS.iWarningCode := 1;
END_IF

IF Lynus_Standards.GVL_Energy.stNumberOfDevices.diNumberOfECS > Constants_Energy.diMaxNumberOfElectricChargingStations THEN fbCS.iErrorCode := 1;
ELSIF bErrorExt THEN fbCS.iErrorCode := 0;
END_IF        	
	
(*------------------------------------------------------------------Logic----------------------------------------------------------------------------*)

//Calcualte the total SOC if we have more then 1 battery in our system
diNumberOfActiveBatterys := 0;
	dwSumSOC := 0;
		FOR liLPBatteryData := 1 TO Constants_Energy.diMaxNumberOfBatterys BY 1 DO
			IF Lynus_Standards.GVL_Energy.stDataOfBatterys[diNrOfEMS_IN,liLPBatteryData].bEnabled THEN diNumberOfActiveBatterys := diNumberOfActiveBatterys + 1; END_IF
				dwSumSOC := dwSumSOC + Lynus_Standards.GVL_Energy.stDataOfBatterys[diNrOfEMS_IN,liLPBatteryData].dwSOC;
		END_FOR
	
IF diNumberOfActiveBatterys > 0 THEN
	fbCS.dwBatterySOC := DINT_TO_DWORD(DWORD_TO_DINT(dwSumSOC) / diNumberOfActiveBatterys);
ELSE
	fbCS.dwBatterySOC := 100;	//When we have no battery in the ems system
END_IF

//Check if one or more Batterysystems or batteryinverter make island mode
diNumberOfBatteryInverterInEPO := 0;
	FOR liLPInEPO := 1 TO Constants_Energy.diMaxNumberOfBatteryInverters BY 1 DO
		IF Lynus_Standards.GVL_Energy.stDataOfBatteryInverters[diNrOfEMS_IN,liLPInEPO].bWorkOnIslandMode THEN fbCS.bEPOIsActive := TRUE; diNumberOfBatteryInverterInEPO := diNumberOfBatteryInverterInEPO + 1; END_IF
	END_FOR 
		IF diNumberOfBatteryInverterInEPO <= 0 THEN fbCS.bEPOIsActive := FALSE; END_IF

//Digital input for external lock signal
fbDIExternalLock(bInvers:= FALSE, bSignal=> );

//Car SOC, charging Time and Mode 3
fbCS.arrSOCCar[1] := 0;
fbCS.arrSOCCar[2] := 0;
fbCS.arrSOCCar[3] := 0;
fbCS.arrSOCCar[4] := 0;
	fbCS.arrSocketChargingTimeInput[1] := 0;
	fbCS.arrSocketChargingTimeInput[2] := 0;
	fbCS.arrSocketChargingTimeInput[3] := 0;
	fbCS.arrSocketChargingTimeInput[4] := 0;
		fbCS.arrSocketMode3StateECS[1] := '';
		fbCS.arrSocketMode3StateECS[2] := '';
		fbCS.arrSocketMode3StateECS[3] := '';
		fbCS.arrSocketMode3StateECS[4] := '';
	
//Functionblock ECS
fbCS(
	bEnable:= bEnable AND NOT timDissableFunctions.Q, 
	bError:= , 
	bEPOIsActive:= , 
	bExternalLock:= fbDIExternalLock.bSignal, 
	bCarConnected:= bCarConnectedExt, 
	bWriteWithDelay:= TRUE, 
	bCalculateEnergySession:= ,
	iErrorCode:= , 
	iWarningCode:= , 
	arrSocketChargingTimeInput:= , 
	arrSOCCar:= , 
	dwBatterySOC:= , 
	lrTotalCounterEnergy_Consumption:= , 
	lrTotalCounterEnergy_Production:= , 
	lrCounterEnergyT1_Consumption:= , 
	lrCounterEnergyT2_Consumption:= , 
	lrCounterEnergyT1_Production:= , 
	lrCounterEnergyT2_Production:= , 
	lrTotalPowerECS:= , 
	arrSocketEnergySession:= ,
	rTargetPower:= Lynus_Standards.GVL_Energy.stDataElectricChargingStations[diNrOfEMS_IN,diNrOfECS_OUT].rTargetPowerEMS, 
	rSupplyVoltage:= 692, 
	rMinCurrent:= 0, 
	tTimDelayOutput:= T#5S, 
	tDelayError:= T#5S,
	arrSocketMode3StateECS:= ,
	arrSocketPowerECS:= ,
	stSetupECS:= stSetupECS, 
	stDataECSOut=> , 
	stDataECSOutDelay=> stDataECS);	
	
(*-------------------------------------------------------------------------Output----------------------------------------------------------------------*)

IF bNoLinear THEN 
	fbInterpolation.rXInputValue := (stSetupECS.rMaxPower * fbCS.stDataECSOut.rTargetPower) / 100; 
		fbInterpolation.arrYIntermediateValues[1] := 10;
			fbInterpolation.arrYIntermediateValues[2] := 20;
				fbInterpolation.arrYIntermediateValues[3] := 30;
					fbInterpolation.arrYIntermediateValues[4] := 40;
						fbInterpolation.arrYIntermediateValues[5] := 50;
	fbInterpolation.arrYIntermediateValues[6] := 60;
		fbInterpolation.arrYIntermediateValues[7] := 70;
			fbInterpolation.arrYIntermediateValues[8] := 80;
				fbInterpolation.arrYIntermediateValues[9] := 90;
					fbInterpolation.arrYIntermediateValues[10] := 100;
	fbInterpolation(rXInputValue:=, arrXIntermediateValues:= arrTableOfInterpolationPoints, arrYIntermediateValues:=, rYOutputValue=> );
END_IF

IF bNoLinear THEN 
	fbAOCS.rSignal := fbInterpolation.rYOutputValue;
	//Target Power, to use this on a external Function
	rTargetPowerForExtFunc := fbInterpolation.rYOutputValue;
	rTargetChargCurrentForExtFunc := (fbCS.stDataECSOut.rTargetChargeCurrent * rTargetPowerForExtFunc) / 100; 
ELSE
	fbAOCS.rSignal := fbCS.stDataECSOut.rTargetPower;
	//Target Power, to use this on a external Function
	rTargetPowerForExtFunc := fbCS.stDataECSOut.rTargetPower;
	rTargetChargCurrentForExtFunc := fbCS.stDataECSOut.rTargetChargeCurrent;
END_IF

fbAOCS(
	rYMinTerminalValue:= 0, 
	rXMinInputSignal:= 0, 
	rYMaxTerminalValue:= 32767, 
	rXMaxInputSignal:= 100, 
	rSignal:= , 
	usiState=> );
							
(*-----------------------------------------------------------Handle data to Global structure for electric charging stations-----------------------------------------------------------------*)

//Delte al old Data on GVL after a online change or change on the variable diNrOfEMS_IDOD
IF diNrOfEMS_IN <> diNrOfEMS_IN_CP AND iStateGVLData = 0 THEN iStateGVLData := 10; END_IF 

CASE iStateGVLData OF
	
	0://Init Step
		byWaitInStep := 0;
			diCounterForGVL := 1;
	
	1://Wait for 4 Steps before clean al Data on GVL
		byWaitInStep := byWaitInStep + 1;
			IF byWaitInStep >= 4 AND fbNumberDevice.bNumberIsCalculatet THEN iStateGVLData := 2; END_IF
				//To much Devices, back to the Init step
				IF byWaitInStep >= 4 AND NOT fbNumberDevice.bNumberIsCalculatet THEN iStateGVLData := 0; END_IF	
			
	2://Clear all Data in GVL
		FOR diLPForGVL := 1 TO Constants_Energy.diMaxNumberOfEMS BY 1 DO 
			Lynus_Standards.GVL_Energy.stDataElectricChargingStations[diLPForGVL,diCounterForGVL].bEnabled := FALSE;
				Lynus_Standards.GVL_Energy.stDataElectricChargingStations[diLPForGVL,diCounterForGVL].bIsControllable := FALSE;
					Lynus_Standards.GVL_Energy.stDataElectricChargingStations[diLPForGVL,diCounterForGVL].byErrorWarning := 0;
						Lynus_Standards.GVL_Energy.stDataElectricChargingStations[diLPForGVL,diCounterForGVL].byPriority := 0;
							Lynus_Standards.GVL_Energy.stDataElectricChargingStations[diLPForGVL,diCounterForGVL].lrPower := 0;
								Lynus_Standards.GVL_Energy.stDataElectricChargingStations[diLPForGVL,diCounterForGVL].lrPowerConsumption := 0;
									Lynus_Standards.GVL_Energy.stDataElectricChargingStations[diLPForGVL,diCounterForGVL].lrPowerProduction := 0;
										Lynus_Standards.GVL_Energy.stDataElectricChargingStations[diLPForGVL,diCounterForGVL].rMaxPower := 0;
											Lynus_Standards.GVL_Energy.stDataElectricChargingStations[diLPForGVL,diCounterForGVL].byElectricFuseLine := 0;
												//Set also the target value from ems back here to 0 and not in EMS function because EMS is in Standy when we have a online change (Problem when we delete a ems function and make a online change)
												Lynus_Standards.GVL_Energy.stDataElectricChargingStations[diLPForGVL,diCounterForGVL].rTargetPowerEMS := 0;	
		END_FOR
			diCounterForGVL := diCounterForGVL + 1;
				diCounterForGVL := LIMIT(0,diCounterForGVL,Constants_Energy.diMaxNumberOfElectricChargingStations);
					//Back to the init step
					IF diCounterForGVL >= Constants_Energy.diMaxNumberOfElectricChargingStations THEN iStateGVLData := 0; END_IF

	10://Clear old Data on GVL 		
		Lynus_Standards.GVL_Energy.stDataElectricChargingStations[diNrOfEMS_IN_CP,diNrOfECS_OUT].bEnabled := FALSE;
			Lynus_Standards.GVL_Energy.stDataElectricChargingStations[diNrOfEMS_IN_CP,diNrOfECS_OUT].bIsControllable := FALSE;
				Lynus_Standards.GVL_Energy.stDataElectricChargingStations[diNrOfEMS_IN_CP,diNrOfECS_OUT].byErrorWarning := 0;
					Lynus_Standards.GVL_Energy.stDataElectricChargingStations[diNrOfEMS_IN_CP,diNrOfECS_OUT].byPriority := 0;
						Lynus_Standards.GVL_Energy.stDataElectricChargingStations[diNrOfEMS_IN_CP,diNrOfECS_OUT].lrPower := 0;
							Lynus_Standards.GVL_Energy.stDataElectricChargingStations[diNrOfEMS_IN_CP,diNrOfECS_OUT].lrPowerConsumption := 0;
								Lynus_Standards.GVL_Energy.stDataElectricChargingStations[diNrOfEMS_IN_CP,diNrOfECS_OUT].lrPowerProduction := 0;
									Lynus_Standards.GVL_Energy.stDataElectricChargingStations[diNrOfEMS_IN_CP,diNrOfECS_OUT].rMaxPower := 0;
										Lynus_Standards.GVL_Energy.stDataElectricChargingStations[diNrOfEMS_IN_CP,diNrOfECS_OUT].byElectricFuseLine := 0;
									
		diNrOfEMS_IN_CP := diNrOfEMS_IN;
			//Back to the init step
			iStateGVLData := 0;

END_CASE 	 

IF diNrOfECS_OUT > 0 AND fbNumberDevice.bNumberIsCalculatet AND diNrOfEMS_IN > 0 THEN
	Lynus_Standards.GVL_Energy.stDataElectricChargingStations[diNrOfEMS_IN,diNrOfECS_OUT].bEnabled := fbCS.stDataECSOut.bEnabled;
		Lynus_Standards.GVL_Energy.stDataElectricChargingStations[diNrOfEMS_IN,diNrOfECS_OUT].bIsControllable := TRUE;
			Lynus_Standards.GVL_Energy.stDataElectricChargingStations[diNrOfEMS_IN,diNrOfECS_OUT].byErrorWarning := fbCS.stDataECSOut.byErrorWarning;
				Lynus_Standards.GVL_Energy.stDataElectricChargingStations[diNrOfEMS_IN,diNrOfECS_OUT].byPriority := fbCS.stDataECSOut.byPriority;
					Lynus_Standards.GVL_Energy.stDataElectricChargingStations[diNrOfEMS_IN,diNrOfECS_OUT].lrPower := fbCS.stDataECSOut.lrTotalPower;
						Lynus_Standards.GVL_Energy.stDataElectricChargingStations[diNrOfEMS_IN,diNrOfECS_OUT].lrPowerConsumption := fbCS.stDataECSOut.lrTotalPowerConsumption;
							Lynus_Standards.GVL_Energy.stDataElectricChargingStations[diNrOfEMS_IN,diNrOfECS_OUT].lrPowerProduction := fbCS.stDataECSOut.lrTotalPowerProduction;
								Lynus_Standards.GVL_Energy.stDataElectricChargingStations[diNrOfEMS_IN,diNrOfECS_OUT].rMaxPower := fbCS.stDataECSOut.rMaxPower;	
									Lynus_Standards.GVL_Energy.stDataElectricChargingStations[diNrOfEMS_IN,diNrOfECS_OUT].byElectricFuseLine := byElectricFuseLine;	
END_IF 
		
(*----------------------------------------------------------Save persistent data----------------------------------------------------------------*)

arrPD[1](lrValue:= BOOL_TO_LREAL(bEnable), bEventBasedActive=> );
arrPD[2](lrValue:= BOOL_TO_LREAL(bPowerDataInvers), bEventBasedActive=> );
arrPD[3](lrValue:= DINT_TO_LREAL(diNrOfEMS_IN), bEventBasedActive=> );
arrPD[4](lrValue:= DINT_TO_LREAL(diNrOfEM_IN_CS), bEventBasedActive=> );
arrPD[5](lrValue:= BOOL_TO_LREAL(stSetupECS.bManualyOn), bEventBasedActive=> );
arrPD[6](lrValue:= BOOL_TO_LREAL(stSetupECS.bOnEmergPowerOff), bEventBasedActive=> );
arrPD[7](lrValue:= BYTE_TO_LREAL(stSetupECS.byCSMinPower), bEventBasedActive=> );
arrPD[8](lrValue:= BYTE_TO_LREAL(stSetupECS.byDisableSOC), bEventBasedActive=> );
arrPD[9](lrValue:= BYTE_TO_LREAL(stSetupECS.byEnableSOC), bEventBasedActive=> );
arrPD[10](lrValue:= BYTE_TO_LREAL(stSetupECS.byManualyTargetPower), bEventBasedActive=> );
arrPD[11](lrValue:= BYTE_TO_LREAL(stSetupECS.byPriority), bEventBasedActive=> );
arrPD[12](lrValue:= REAL_TO_LREAL(stSetupECS.rMaxPower), bEventBasedActive=> );
arrPD[13](lrValue:= DINT_TO_LREAL(diNrOfEMS_IN_CP), bEventBasedActive=> );
arrPD[14](lrValue:= BOOL_TO_LREAL(bNoLinear), bEventBasedActive=> );
arrPD[15](lrValue:= REAL_TO_LREAL(arrTableOfInterpolationPoints[1]), bEventBasedActive=> );
arrPD[16](lrValue:= REAL_TO_LREAL(arrTableOfInterpolationPoints[2]), bEventBasedActive=> );
arrPD[17](lrValue:= REAL_TO_LREAL(arrTableOfInterpolationPoints[3]), bEventBasedActive=> );
arrPD[18](lrValue:= REAL_TO_LREAL(arrTableOfInterpolationPoints[4]), bEventBasedActive=> );
arrPD[19](lrValue:= REAL_TO_LREAL(arrTableOfInterpolationPoints[5]), bEventBasedActive=> );
arrPD[20](lrValue:= REAL_TO_LREAL(arrTableOfInterpolationPoints[6]), bEventBasedActive=> );
arrPD[21](lrValue:= REAL_TO_LREAL(arrTableOfInterpolationPoints[7]), bEventBasedActive=> );
arrPD[22](lrValue:= REAL_TO_LREAL(arrTableOfInterpolationPoints[8]), bEventBasedActive=> );
arrPD[23](lrValue:= REAL_TO_LREAL(arrTableOfInterpolationPoints[9]), bEventBasedActive=> );
arrPD[24](lrValue:= REAL_TO_LREAL(arrTableOfInterpolationPoints[10]), bEventBasedActive=> );
arrPD[25](lrValue:= BYTE_TO_LREAL(byElectricFuseLine), bEventBasedActive=> );

END_FUNCTION_BLOCK

// ---- FBs/Electric Charging Station/OnOff/FB_ECS_OnOff.TcPOU
FUNCTION_BLOCK FB_ECS_OnOff
VAR_INPUT PERSISTENT
	bEnable									: BOOL;											//{#lynus.ag#()} //Enable the Fuctionblock and his logic
	bPowerDataInvers						: BOOL;											//With True its possible to invert all received power data from the electric meter
	byElectricFuseLine						: BYTE; 										//Electric Fuse Line on wich the ECS is connected => 1 2 3 (If 0 then this charging station is not connected to a Electric Fuse Line)
	diNrOfEMS_IN							: DINT;											//Number of EMS what control this Device.
	diNrOfEM_IN_CS							: DINT;											//Number of the electric meter for incoming power data. (Power Data for this Device)
	stSetupECS								: ST_Setup_ECS;									//{#lynus.ag#()} //Setup charging station
END_VAR
VAR_INPUT
END_VAR
VAR_OUTPUT
	stDataECS								: ST_ECS_Output;								//{#lynus.ag#()} //Electric charging station output data
	diNrOfECS_OUT							: DINT;											//Active Number from the Electric charging Function for using on other functions
	rTargetPowerForExtFunc					: REAL;											//Target Power from 0% to +100% to use on a external Function
END_VAR
VAR
	{attribute 'hide'}
	fbCS									: FB_ElectricChargingStation;					//Function block for electric charging station
	{attribute 'hide'}
	fbNumberDevice							: FB_NumberOfDevice;							//Function block to calcualte the number of the Device
	fbDIExternalLock						: FB_XL1XXX_DI;									//Digital Input from external loock signal
	fbDOOnOffCS								: FB_XL2XXX_DO;									//Digital Output to swtich on and off the charging station
	{attribute 'hide'}
	timDissableFunctions					: TON;											//Timer to dissable the Function after Lynus_Standards.Constants_General.tTimeDissableLynusFunctions Days without connection to the Lynus Cloud
	{attribute 'hide'}
	timResetConnectionOnGVL					: TON;											//Timer to try reset the connection Flag on the GVL. (When somebody delete the Connection Function and make only a onlinechange)
	{attribute 'hide'}
	arrPD									: ARRAY[1..14] OF FB_PersistentData_Number;		//Function to save persistent data 
	{attribute 'hide'}
	byWaitInStep							: BYTE;											//Wait in Step before start to clean data on PLC
	{attribute 'hide'}
	iStateGVLData							: INT;											//State machine to handle the data on the GVL
	{attribute 'hide'}
	diNumberOfActiveBatterys				: DINT;											//Number of active batterys
	{attribute 'hide'}
	diNumberOfBatteryInverterInEPO			: DINT;											//Number of battery inverters that work in Emergency Power operation 
	{attribute 'hide'}
	diCounterForGVL							: DINT;											//Counter to clean old data on GVL
	{attribute 'hide'}
	diLPForGVL								: DINT;											//Loop to clean old data on GVL
	{attribute 'hide'}
	dwSumSOC								: DWORD;										//Sum of the SOC from all batterys	
	{attribute 'hide'}
	liLPBatteryData							: LINT;											//Loop to check some data from batterys
	{attribute 'hide'}
	liLPInEPO								: LINT;											//Loop to check if 1 or more battery inverters build a island grid
END_VAR
VAR PERSISTENT
	{attribute 'conditionalshow'}
	diNrOfEMS_IN_CP							: DINT;											//Number of EMS what control this Device to compare with the original
END_VAR

//Creator : Kai Ebensperger
//Company : Lynus AG
//Date : 19.05.2021
//Version : 1.0.0.0

//With this function block its possible to switch on and off a charging station
//The output signal to switch on and off is a digital output signal
//With this function block its not possible to control the CS with a target power value because we didn't have a active communication to the CS
//With the Nr from the Electric Meter its possible to send the data fromt the electric meter directly to the CS function to display it

//NOTE for diNr.....Designation => 
//_IN = Here Data come in from other Functions or go out to other functions about the GVL
//_OUT = Here Data go out to other functions about the GVL

(*------------------------------------------------------------Limits----------------------------------------------------------------------------------*)

diNrOfEMS_IN := LIMIT(0,diNrOfEMS_IN,Constants_Energy.diMaxNumberOfEMS);
	diNrOfEM_IN_CS := LIMIT(0,diNrOfEM_IN_CS,Constants_Energy.diMaxNumberOfElectricMeters);
		byElectricFuseLine := LIMIT(0,byElectricFuseLine,30);	
			
(*------------------------------------------------------------------Power Data----------------------------------------------------------------------------*)

//Energy Session Input data
fbCS.bCalculateEnergySession := FALSE;
fbCS.arrSocketPowerECS[1] := 0;
fbCS.arrSocketPowerECS[2] := 0;
fbCS.arrSocketPowerECS[3] := 0;
fbCS.arrSocketPowerECS[4] := 0;
fbCS.arrSocketEnergySession[1] := 0;
fbCS.arrSocketEnergySession[2] := 0;
fbCS.arrSocketEnergySession[3] := 0;
fbCS.arrSocketEnergySession[4] := 0;

IF NOT bPowerDataInvers THEN
	fbCS.lrCounterEnergyT1_Consumption := Lynus_Standards.GVL_Energy.stDataElectricMeters[diNrOfEM_IN_CS].lrCounterEnergyT1_Production * 1000;
	fbCS.lrCounterEnergyT2_Consumption := Lynus_Standards.GVL_Energy.stDataElectricMeters[diNrOfEM_IN_CS].lrCounterEnergyT2_Production * 1000;
	fbCS.lrCounterEnergyT1_Production := Lynus_Standards.GVL_Energy.stDataElectricMeters[diNrOfEM_IN_CS].lrCounterEnergyT1_Consumption * 1000;
	fbCS.lrCounterEnergyT2_Production := Lynus_Standards.GVL_Energy.stDataElectricMeters[diNrOfEM_IN_CS].lrCounterEnergyT1_Consumption * 1000;
	fbCS.lrTotalCounterEnergy_Consumption := Lynus_Standards.GVL_Energy.stDataElectricMeters[diNrOfEM_IN_CS].lrTotalCounterEnergy_Production * 1000;
	fbCS.lrTotalCounterEnergy_Production := Lynus_Standards.GVL_Energy.stDataElectricMeters[diNrOfEM_IN_CS].lrTotalCounterEnergy_Consumption * 1000;
		fbCS.lrTotalPowerECS := (Lynus_Standards.GVL_Energy.stDataElectricMeters[diNrOfEM_IN_CS].lrPower * 1000) * - 1;
ELSE
	fbCS.lrCounterEnergyT1_Consumption := Lynus_Standards.GVL_Energy.stDataElectricMeters[diNrOfEM_IN_CS].lrCounterEnergyT1_Consumption * 1000;
	fbCS.lrCounterEnergyT2_Consumption := Lynus_Standards.GVL_Energy.stDataElectricMeters[diNrOfEM_IN_CS].lrCounterEnergyT2_Consumption * 1000;
	fbCS.lrCounterEnergyT1_Production := Lynus_Standards.GVL_Energy.stDataElectricMeters[diNrOfEM_IN_CS].lrCounterEnergyT1_Production * 1000;
	fbCS.lrCounterEnergyT2_Production := Lynus_Standards.GVL_Energy.stDataElectricMeters[diNrOfEM_IN_CS].lrCounterEnergyT2_Production * 1000;
	fbCS.lrTotalCounterEnergy_Consumption := Lynus_Standards.GVL_Energy.stDataElectricMeters[diNrOfEM_IN_CS].lrTotalCounterEnergy_Consumption * 1000;
	fbCS.lrTotalCounterEnergy_Production := Lynus_Standards.GVL_Energy.stDataElectricMeters[diNrOfEM_IN_CS].lrTotalCounterEnergy_Production * 1000;
		fbCS.lrTotalPowerECS := Lynus_Standards.GVL_Energy.stDataElectricMeters[diNrOfEM_IN_CS].lrPower * 1000;
END_IF

(*-------------------------------------------------------------Calcualte the number of ECS---------------------------------------------------------------*)

fbNumberDevice(
	diActualNumberOfDevices:= Lynus_Standards.GVL_Energy.stNumberOfDevices.diNumberOfECS, 
	diMaxNumberOfDevices:= Constants_Energy.diMaxNumberOfElectricChargingStations, 
	udiCounterOnlineChange:= TwinCAT_SystemInfoVarList._AppInfo.OnlineChangeCnt, 
	bNumberIsCalculatet=> , 
	bFPNumberIsCalculatet=> , 
	bOnlineChange=> , 
	diNumberForThisDevice=> diNrOfECS_OUT, 
	diNumberOfTotalDevices=> );

//Write new Numer on GVL
IF fbNumberDevice.bFPNumberIsCalculatet THEN
	Lynus_Standards.GVL_Energy.stNumberOfDevices.diNumberOfECS := fbNumberDevice.diNumberOfTotalDevices;	
END_IF 

//Delete old Number on GVL
IF fbNumberDevice.bOnlineChange THEN 
	Lynus_Standards.GVL_Energy.stNumberOfDevices.diNumberOfECS := diNrOfECS_OUT;	
		iStateGVLData := 1; 
END_IF

(*-------------------------------------------------------------Service from Backend is ready and check the connection to backen for dissabel/enable Function---------------------------------------------------------------*)

//Try to reset the variable for connection on the GVL. When all is normal then the Lynus Mqtt connection function set this variable to true in the next cycle
//When we have no connection to the backend then after Lynus_Standards.Constants_General.tTimeDissableLynusFunctions days the Function is dissabled with all of his functionalities
timResetConnectionOnGVL(IN:= NOT timResetConnectionOnGVL.Q, PT:= T#1H, Q=> , ET=> );
	IF timResetConnectionOnGVL.Q THEN Lynus_Standards.GVL_Communicator.bStateConnectionToEnableFunctions := FALSE; END_IF
		IF NOT Lynus_Standards.GVL_Communicator.bStateConnectionToEnableFunctions THEN timDissableFunctions.IN := TRUE; ELSE timDissableFunctions.IN := FALSE; END_IF  
			timDissableFunctions(IN:= , PT:= Lynus_Standards.Constants_General.tTimeDissableLynusFunctions, Q=> , ET=> );


(*------------------------------------------------------------------Error and Warning----------------------------------------------------------------------------*)	

IF timDissableFunctions.Q THEN fbCS.bWarning := TRUE; fbCS.iWarningCode := 0; ELSE fbCS.bWarning := FALSE; END_IF   
	IF Lynus_Standards.GVL_Energy.stNumberOfDevices.diNumberOfECS > Constants_Energy.diMaxNumberOfElectricChargingStations THEN 
		fbCS.bError := TRUE;
			fbCS.iErrorCode := 1; 
	ELSE 
		fbCS.bError := FALSE;
			fbCS.iErrorCode := 0; 
	END_IF

(*------------------------------------------------------------------Logic----------------------------------------------------------------------------*)

//Calcualte the total SOC if we have more then 1 battery in our system
diNumberOfActiveBatterys := 0;
	dwSumSOC := 0;
		FOR liLPBatteryData := 1 TO Constants_Energy.diMaxNumberOfBatterys BY 1 DO
			IF Lynus_Standards.GVL_Energy.stDataOfBatterys[diNrOfEMS_IN,liLPBatteryData].bEnabled THEN diNumberOfActiveBatterys := diNumberOfActiveBatterys + 1; END_IF
				dwSumSOC := dwSumSOC + Lynus_Standards.GVL_Energy.stDataOfBatterys[diNrOfEMS_IN,liLPBatteryData].dwSOC;
		END_FOR
	
IF diNumberOfActiveBatterys > 0 THEN
	fbCS.dwBatterySOC := DINT_TO_DWORD(DWORD_TO_DINT(dwSumSOC) / diNumberOfActiveBatterys);
ELSE
	fbCS.dwBatterySOC := 100;	//When we have no battery in the ems system
END_IF

//Check if one or more Batterysystems or batteryinverter make island mode
diNumberOfBatteryInverterInEPO := 0;
	FOR liLPInEPO := 1 TO Constants_Energy.diMaxNumberOfBatteryInverters BY 1 DO
		IF Lynus_Standards.GVL_Energy.stDataOfBatteryInverters[diNrOfEMS_IN,liLPInEPO].bWorkOnIslandMode THEN fbCS.bEPOIsActive := TRUE; diNumberOfBatteryInverterInEPO := diNumberOfBatteryInverterInEPO + 1; END_IF
	END_FOR 
		IF diNumberOfBatteryInverterInEPO <= 0 THEN fbCS.bEPOIsActive := FALSE; END_IF

//Digital input for external lock signal
fbDIExternalLock(bInvers:= FALSE, bSignal=> );

//Functionblock ECS
fbCS.stSetupECS.bManualyOn := stSetupECS.bManualyOn;
	IF fbCS.stSetupECS.bManualyOn THEN fbCS.stSetupECS.byManualyTargetPower := 100; ELSE fbCS.stSetupECS.byManualyTargetPower := 0; END_IF
		fbCS.stSetupECS.bOnEmergPowerOff := stSetupECS.bOnEmergPowerOff;
			fbCS.stSetupECS.byDisableSOC := stSetupECS.byDisableSOC;
				fbCS.stSetupECS.byEnableSOC := stSetupECS.byEnableSOC;
					fbCS.stSetupECS.byCSMinPower := stSetupECS.byCSMinPower;
						fbCS.stSetupECS.byPriority := stSetupECS.byPriority;
							fbCS.stSetupECS.rMaxPower := stSetupECS.rMaxPower;

//Car SOC, charging Time and Mode 3
fbCS.arrSOCCar[1] := 0;
fbCS.arrSOCCar[2] := 0;
fbCS.arrSOCCar[3] := 0;
fbCS.arrSOCCar[4] := 0;
	fbCS.arrSocketChargingTimeInput[1] := 0;
	fbCS.arrSocketChargingTimeInput[2] := 0;
	fbCS.arrSocketChargingTimeInput[3] := 0;
	fbCS.arrSocketChargingTimeInput[4] := 0;
		fbCS.arrSocketMode3StateECS[1] := '';
		fbCS.arrSocketMode3StateECS[2] := '';
		fbCS.arrSocketMode3StateECS[3] := '';
		fbCS.arrSocketMode3StateECS[4] := '';							
							
fbCS(
	bEnable:= bEnable AND NOT timDissableFunctions.Q, 
	bError:= , 
	bEPOIsActive:= , 
	bExternalLock:= fbDIExternalLock.bSignal, 
	bCarConnected:= FALSE, 
	bWriteWithDelay:= TRUE, 
	bCalculateEnergySession:= ,
	iErrorCode:= , 
	iWarningCode:= , 
	arrSocketChargingTimeInput:= , 
	arrSOCCar:= , 
	dwBatterySOC:= , 
	lrTotalCounterEnergy_Consumption:= , 
	lrTotalCounterEnergy_Production:= , 
	lrCounterEnergyT1_Consumption:= , 
	lrCounterEnergyT2_Consumption:= , 
	lrCounterEnergyT1_Production:= , 
	lrCounterEnergyT2_Production:= , 
	lrTotalPowerECS:= ,
	arrSocketEnergySession:= , 
	rTargetPower:= Lynus_Standards.GVL_Energy.stDataElectricChargingStations[diNrOfEMS_IN,diNrOfECS_OUT].rTargetPowerEMS, 
	rSupplyVoltage:= 692, 
	rMinCurrent:= 0, 
	tTimDelayOutput:= T#5S, 
	tDelayError:= T#5S,
	arrSocketMode3StateECS:= ,
	arrSocketPowerECS:= ,
	stSetupECS:= , 
	stDataECSOut=> , 
	stDataECSOutDelay=> stDataECS);

//Target Power, to use this on a external Function
rTargetPowerForExtFunc := fbCS.stDataECSOut.rTargetPower;	
	
(*-------------------------------------------------------------------------Output----------------------------------------------------------------------*)

fbDOOnOffCS(bInvers:= FALSE, bSignal:= fbCS.stDataECSOut.bOutputOnOff);
							
(*-----------------------------------------------------------Handle data to Global structure for electric charging stations-----------------------------------------------------------------*)

//Delte al old Data on GVL after a online change or change on the variable diNrOfEMS_IDOD
IF diNrOfEMS_IN <> diNrOfEMS_IN_CP AND iStateGVLData = 0 THEN iStateGVLData := 10; END_IF 

CASE iStateGVLData OF
	
	0://Init Step
		byWaitInStep := 0;
			diCounterForGVL := 1;
	
	1://Wait for 4 Steps before clean al Data on GVL
		byWaitInStep := byWaitInStep + 1;
			IF byWaitInStep >= 4 AND fbNumberDevice.bNumberIsCalculatet THEN iStateGVLData := 2; END_IF
				//To much Devices, back to the Init step
				IF byWaitInStep >= 4 AND NOT fbNumberDevice.bNumberIsCalculatet THEN iStateGVLData := 0; END_IF	
			
	2://Clear all Data in GVL
		FOR diLPForGVL := 1 TO Constants_Energy.diMaxNumberOfEMS BY 1 DO 
			Lynus_Standards.GVL_Energy.stDataElectricChargingStations[diLPForGVL,diCounterForGVL].bEnabled := FALSE;
				Lynus_Standards.GVL_Energy.stDataElectricChargingStations[diLPForGVL,diCounterForGVL].bIsControllable := FALSE;
					Lynus_Standards.GVL_Energy.stDataElectricChargingStations[diLPForGVL,diCounterForGVL].byErrorWarning := 0;
						Lynus_Standards.GVL_Energy.stDataElectricChargingStations[diLPForGVL,diCounterForGVL].byPriority := 0;
							Lynus_Standards.GVL_Energy.stDataElectricChargingStations[diLPForGVL,diCounterForGVL].lrPower := 0;
								Lynus_Standards.GVL_Energy.stDataElectricChargingStations[diLPForGVL,diCounterForGVL].lrPowerConsumption := 0;
									Lynus_Standards.GVL_Energy.stDataElectricChargingStations[diLPForGVL,diCounterForGVL].lrPowerProduction := 0;
										Lynus_Standards.GVL_Energy.stDataElectricChargingStations[diLPForGVL,diCounterForGVL].rMaxPower := 0;
											Lynus_Standards.GVL_Energy.stDataElectricChargingStations[diLPForGVL,diCounterForGVL].byElectricFuseLine := 0;
												//Set also the target value from ems back here to 0 and not in EMS function because EMS is in Standy when we have a online change (Problem when we delete a ems function and make a online change)
												Lynus_Standards.GVL_Energy.stDataElectricChargingStations[diLPForGVL,diCounterForGVL].rTargetPowerEMS := 0;	
		END_FOR
			diCounterForGVL := diCounterForGVL + 1;
				diCounterForGVL := LIMIT(0,diCounterForGVL,Constants_Energy.diMaxNumberOfElectricChargingStations);
					//Back to the init step
					IF diCounterForGVL >= Constants_Energy.diMaxNumberOfElectricChargingStations THEN iStateGVLData := 0; END_IF

	10://Clear old Data on GVL 		
		Lynus_Standards.GVL_Energy.stDataElectricChargingStations[diNrOfEMS_IN_CP,diNrOfECS_OUT].bEnabled := FALSE;
			Lynus_Standards.GVL_Energy.stDataElectricChargingStations[diNrOfEMS_IN_CP,diNrOfECS_OUT].bIsControllable := FALSE;
				Lynus_Standards.GVL_Energy.stDataElectricChargingStations[diNrOfEMS_IN_CP,diNrOfECS_OUT].byErrorWarning := 0;
					Lynus_Standards.GVL_Energy.stDataElectricChargingStations[diNrOfEMS_IN_CP,diNrOfECS_OUT].byPriority := 0;
						Lynus_Standards.GVL_Energy.stDataElectricChargingStations[diNrOfEMS_IN_CP,diNrOfECS_OUT].lrPower := 0;
							Lynus_Standards.GVL_Energy.stDataElectricChargingStations[diNrOfEMS_IN_CP,diNrOfECS_OUT].lrPowerConsumption := 0;
								Lynus_Standards.GVL_Energy.stDataElectricChargingStations[diNrOfEMS_IN_CP,diNrOfECS_OUT].lrPowerProduction := 0;
									Lynus_Standards.GVL_Energy.stDataElectricChargingStations[diNrOfEMS_IN_CP,diNrOfECS_OUT].rMaxPower := 0;
										Lynus_Standards.GVL_Energy.stDataElectricChargingStations[diNrOfEMS_IN_CP,diNrOfECS_OUT].byElectricFuseLine := 0;
									
		diNrOfEMS_IN_CP := diNrOfEMS_IN;
			//Back to the init step
			iStateGVLData := 0;

END_CASE 	 

IF diNrOfECS_OUT > 0 AND fbNumberDevice.bNumberIsCalculatet AND diNrOfEMS_IN > 0 THEN
	Lynus_Standards.GVL_Energy.stDataElectricChargingStations[diNrOfEMS_IN,diNrOfECS_OUT].bEnabled := fbCS.stDataECSOut.bEnabled;
		Lynus_Standards.GVL_Energy.stDataElectricChargingStations[diNrOfEMS_IN,diNrOfECS_OUT].bIsControllable := FALSE;
			Lynus_Standards.GVL_Energy.stDataElectricChargingStations[diNrOfEMS_IN,diNrOfECS_OUT].byErrorWarning := fbCS.stDataECSOut.byErrorWarning;
				Lynus_Standards.GVL_Energy.stDataElectricChargingStations[diNrOfEMS_IN,diNrOfECS_OUT].byPriority := fbCS.stDataECSOut.byPriority;
					Lynus_Standards.GVL_Energy.stDataElectricChargingStations[diNrOfEMS_IN,diNrOfECS_OUT].lrPower := fbCS.stDataECSOut.lrTotalPower;
						Lynus_Standards.GVL_Energy.stDataElectricChargingStations[diNrOfEMS_IN,diNrOfECS_OUT].lrPowerConsumption := fbCS.stDataECSOut.lrTotalPowerConsumption;
							Lynus_Standards.GVL_Energy.stDataElectricChargingStations[diNrOfEMS_IN,diNrOfECS_OUT].lrPowerProduction := fbCS.stDataECSOut.lrTotalPowerProduction;
								Lynus_Standards.GVL_Energy.stDataElectricChargingStations[diNrOfEMS_IN,diNrOfECS_OUT].rMaxPower := fbCS.stDataECSOut.rMaxPower;	
									Lynus_Standards.GVL_Energy.stDataElectricChargingStations[diNrOfEMS_IN,diNrOfECS_OUT].byElectricFuseLine := byElectricFuseLine;
END_IF 
		
(*----------------------------------------------------------Save persistent data----------------------------------------------------------------*)

arrPD[1](lrValue:= BOOL_TO_LREAL(bEnable), bEventBasedActive=> );
arrPD[2](lrValue:= BOOL_TO_LREAL(bPowerDataInvers), bEventBasedActive=> );
arrPD[3](lrValue:= DINT_TO_LREAL(diNrOfEMS_IN), bEventBasedActive=> );
arrPD[4](lrValue:= DINT_TO_LREAL(diNrOfEM_IN_CS), bEventBasedActive=> );
arrPD[5](lrValue:= BOOL_TO_LREAL(stSetupECS.bManualyOn), bEventBasedActive=> );
arrPD[6](lrValue:= BOOL_TO_LREAL(stSetupECS.bOnEmergPowerOff), bEventBasedActive=> );
arrPD[7](lrValue:= BYTE_TO_LREAL(stSetupECS.byCSMinPower), bEventBasedActive=> );
arrPD[8](lrValue:= BYTE_TO_LREAL(stSetupECS.byDisableSOC), bEventBasedActive=> );
arrPD[9](lrValue:= BYTE_TO_LREAL(stSetupECS.byEnableSOC), bEventBasedActive=> );
arrPD[10](lrValue:= BYTE_TO_LREAL(stSetupECS.byManualyTargetPower), bEventBasedActive=> );
arrPD[11](lrValue:= BYTE_TO_LREAL(stSetupECS.byPriority), bEventBasedActive=> );
arrPD[12](lrValue:= REAL_TO_LREAL(stSetupECS.rMaxPower), bEventBasedActive=> );
arrPD[13](lrValue:= DINT_TO_LREAL(diNrOfEMS_IN_CP), bEventBasedActive=> );
arrPD[14](lrValue:= BYTE_TO_LREAL(byElectricFuseLine), bEventBasedActive=> );

END_FUNCTION_BLOCK

// ---- FBs/Electric Heating Element/Linear AO/FB_EHE_Linear_AO.TcPOU
FUNCTION_BLOCK FB_EHE_Linear_AO
VAR_INPUT PERSISTENT
	bEnable									: BOOL;																							//{#lynus.ag#()} //Enable the Fuctionblock and his logic
	bPowerDataInvers						: BOOL;																							//With True its possible to invert all received power data from the electric meter
	bNoLinear								: BOOL;																							//Output Power from the device is not linear. Use the Values from the Table Of Interpolation Points.
	diNrOfEMS_IN							: DINT;																							//Number of EMS what control this Device.
	diNrOfEM_IN_EHE							: DINT;																							//Number of the electric meter for incoming power data. (Power Data for this Device)
	diNrOfTempS_IN							: DINT;																							//Number of the Temperature Sensor for incoming temperature data. (Temperature for the Service wather buffer)
	stSetupEHE								: ST_Setup_EHE := (uiTargetTempOn := 35, uiTargetTempOff := 50, uiTargetTempMax := 62);			//{#lynus.ag#()} //Setup electric heating element
	arrTableOfInterpolationPoints			: ARRAY[1..10] OF REAL;																			//Table Of Interpolation Points. Corresponds to the different power values in the non-linear curve of the device. The last value must correspond to the maximum power.
END_VAR
VAR_INPUT
END_VAR
VAR_OUTPUT
	stDataEHE								: ST_EHE_Output;																				//{#lynus.ag#()} //Electric heating element output data
	diNrOfEHE_OUT							: DINT;																							//Active Number from the Electric heating element for using on other functions
	rTargetPowerForExtFunc					: REAL;																							//Target Power from 0% to +100% to use on a external Function
END_VAR
VAR
	{attribute 'conditionalshow'}
	fbEHE									: FB_ElectricHeatingElement;																	//Function block for electric heating element
	{attribute 'hide'}
	fbNumberDevice							: FB_NumberOfDevice;																			//Function block to calcualte the number of the Device
	{attribute 'hide'}
	fbInterpolation							: FB_Lin_Interpolation;																			//Function for interpolation
	fbDIExternalLock						: FB_XL1XXX_DI;																					//Digital Input from external loock signal
	fbAOEHE									: FB_XL4XXX_AO;																					//Analog Output to swtich on and off and controll the EHE
	{attribute 'hide'}
	timDissableFunctions					: TON;																							//Timer to dissable the Function after Lynus_Standards.Constants_General.tTimeDissableLynusFunctions Days without connection to the Lynus Cloud
	{attribute 'hide'}
	timResetConnectionOnGVL					: TON;																							//Timer to try reset the connection Flag on the GVL. (When somebody delete the Connection Function and make only a onlinechange)
	{attribute 'hide'}
	timGetTime								: TON;																							//Timer to activate the function tho read out the windows system time
	{attribute 'hide'}
	fbGetSystemTime							: NT_GetTime;																					//Function to read out the windows system time on the local plc
	{attribute 'hide'}
	arrPD									: ARRAY[1..42] OF FB_PersistentData_Number;														//Function to save persistent data
	{attribute 'hide'} 
	byLPTargetPowerTo0						: BYTE;																							//Loop to set the target power from the ems and the max power from the settings for arr[2] to arr[10] to 0 because its only a onOff EHE
	{attribute 'hide'}
	byLPGVLSetMaxPower						: BYTE;																							//Loop to send the max power from the EHE to the GVL
	{attribute 'hide'}
	byWaitInStep							: BYTE;																							//Wait in Step before start to clean data on PLC
	{attribute 'hide'}
	iStateGVLData							: INT;																							//State machine to handle the data on the GVL
	{attribute 'hide'}
	diNumberOfActiveBatterys				: DINT;																							//Number of active batterys
	{attribute 'hide'}
	diNumberOfBatteryInverterInEPO			: DINT;																							//Number of battery inverters that work in Emergency Power operation 
	{attribute 'hide'}
	diCounterForGVL							: DINT;																							//Counter to clean old data on GVL
	{attribute 'hide'}
	diLPForGVL								: DINT;																							//Loop to clean old data on GVL
	{attribute 'hide'}
	dwSumSOC								: DWORD;																						//Sum of the SOC from all batterys
	{attribute 'hide'}
	lrGridPower								: LREAL;																						//Grid power in kW
	{attribute 'hide'}
	lrSizeGridConnection					: LREAL;																						//Size of the complete grid connection
	{attribute 'hide'}
	liLPBatteryData							: LINT;																							//Loop to check some data from batterys
	{attribute 'hide'}
	liLPInEPO								: LINT;																							//Loop to check if 1 or more battery inverters build a island grid	
	{attribute 'hide'}
	liLPGridData							: LINT;																							//Loop to check some grid data																				
END_VAR
VAR PERSISTENT
	{attribute 'conditionalshow'}
	diNrOfEMS_IN_CP							: DINT;																							//Number of EMS what control this Device to compare with the original
END_VAR

//Creator : Kai Ebensperger
//Company : Lynus AG
//Date : 19.05.2021
//Version : 1.0.0.0

//With this function block its possible to switch on and off a electric heating element
//The output signal to switch on and off is a analog output signal. (0-10V or 4-20mA)
//With this function block its possible to control the EHE with a target power value over the analog signal. The output signal is linear
//With the Nr from the Electric Meter its possible to send the data fromt the electric meter directly to the EHE function to display it

//NOTE for diNr.....Designation => 
//_IN = Here Data come in from other Functions or go out to other functions about the GVL
//_OUT = Here Data go out to other functions about the GVL

(*------------------------------------------------------------Limits----------------------------------------------------------------------------------*)

diNrOfEMS_IN := LIMIT(0,diNrOfEMS_IN,Constants_Energy.diMaxNumberOfEMS);
	diNrOfEM_IN_EHE := LIMIT(0,diNrOfEM_IN_EHE,Constants_Energy.diMaxNumberOfElectricMeters);
		diNrOfTempS_IN := LIMIT(0,diNrOfTempS_IN,Constants_Sensors.diMaxNumberOfTemperatureSensors);
			
(*------------------------------------------------------------------Power Data----------------------------------------------------------------------------*)

IF NOT bPowerDataInvers THEN
	fbEHE.lrCounterEnergyT1_Consumption := Lynus_Standards.GVL_Energy.stDataElectricMeters[diNrOfEM_IN_EHE].lrCounterEnergyT1_Production * 1000;
	fbEHE.lrCounterEnergyT2_Consumption := Lynus_Standards.GVL_Energy.stDataElectricMeters[diNrOfEM_IN_EHE].lrCounterEnergyT2_Production * 1000;
	fbEHE.lrCounterEnergyT1_Production := Lynus_Standards.GVL_Energy.stDataElectricMeters[diNrOfEM_IN_EHE].lrCounterEnergyT1_Consumption * 1000;
	fbEHE.lrCounterEnergyT2_Production := Lynus_Standards.GVL_Energy.stDataElectricMeters[diNrOfEM_IN_EHE].lrCounterEnergyT1_Consumption * 1000;
	fbEHE.lrTotalCounterEnergy_Consumption := Lynus_Standards.GVL_Energy.stDataElectricMeters[diNrOfEM_IN_EHE].lrTotalCounterEnergy_Production * 1000;
	fbEHE.lrTotalCounterEnergy_Production := Lynus_Standards.GVL_Energy.stDataElectricMeters[diNrOfEM_IN_EHE].lrTotalCounterEnergy_Consumption * 1000;
		fbEHE.lrPowerEHE := (Lynus_Standards.GVL_Energy.stDataElectricMeters[diNrOfEM_IN_EHE].lrPower * 1000) * - 1;
ELSE
	fbEHE.lrCounterEnergyT1_Consumption := Lynus_Standards.GVL_Energy.stDataElectricMeters[diNrOfEM_IN_EHE].lrCounterEnergyT1_Consumption * 1000;
	fbEHE.lrCounterEnergyT2_Consumption := Lynus_Standards.GVL_Energy.stDataElectricMeters[diNrOfEM_IN_EHE].lrCounterEnergyT2_Consumption * 1000;
	fbEHE.lrCounterEnergyT1_Production := Lynus_Standards.GVL_Energy.stDataElectricMeters[diNrOfEM_IN_EHE].lrCounterEnergyT1_Production * 1000;
	fbEHE.lrCounterEnergyT2_Production := Lynus_Standards.GVL_Energy.stDataElectricMeters[diNrOfEM_IN_EHE].lrCounterEnergyT2_Production * 1000;
	fbEHE.lrTotalCounterEnergy_Consumption := Lynus_Standards.GVL_Energy.stDataElectricMeters[diNrOfEM_IN_EHE].lrTotalCounterEnergy_Consumption * 1000;
	fbEHE.lrTotalCounterEnergy_Production := Lynus_Standards.GVL_Energy.stDataElectricMeters[diNrOfEM_IN_EHE].lrTotalCounterEnergy_Production * 1000;
		fbEHE.lrPowerEHE := Lynus_Standards.GVL_Energy.stDataElectricMeters[diNrOfEM_IN_EHE].lrPower * 1000;
END_IF

(*-------------------------------------------------------------Calcualte the number of EHE---------------------------------------------------------------*)

fbNumberDevice(
	diActualNumberOfDevices:= Lynus_Standards.GVL_Energy.stNumberOfDevices.diNumberOfEHE, 
	diMaxNumberOfDevices:= Constants_Energy.diMaxNumberOfElectricHeatingElements, 
	udiCounterOnlineChange:= TwinCAT_SystemInfoVarList._AppInfo.OnlineChangeCnt, 
	bNumberIsCalculatet=> , 
	bFPNumberIsCalculatet=> , 
	bOnlineChange=> , 
	diNumberForThisDevice=> diNrOfEHE_OUT, 
	diNumberOfTotalDevices=> );

//Write new Numer on GVL
IF fbNumberDevice.bFPNumberIsCalculatet THEN
	Lynus_Standards.GVL_Energy.stNumberOfDevices.diNumberOfEHE := fbNumberDevice.diNumberOfTotalDevices;	
END_IF 

//Delete old Number on GVL
IF fbNumberDevice.bOnlineChange THEN 
	Lynus_Standards.GVL_Energy.stNumberOfDevices.diNumberOfEHE := diNrOfEHE_OUT;	
		iStateGVLData := 1; 
END_IF

(*-------------------------------------------------------------Get the local windows system time for this plc---------------------------------------------------------------*)
timGetTime(IN:= bEnable AND NOT timGetTime.Q, PT:= T#30S, Q=> , ET=> );

fbGetSystemTime(
	NETID:= , 
	START:= timGetTime.Q AND NOT fbGetSystemTime.BUSY, 
	TMOUT:= , 
	BUSY=> , 
	ERR=> , 
	ERRID=> , 
	TIMESTR=> );	

fbEHE.stSystemTime.wHour := fbGetSystemTime.TIMESTR.wHour;
	fbEHE.stSystemTime.wMinute := fbGetSystemTime.TIMESTR.wMinute;

(*-------------------------------------------------------------Service from Backend is ready and check the connection to backen for dissabel/enable Function---------------------------------------------------------------*)

//Try to reset the variable for connection on the GVL. When all is normal then the Lynus Mqtt connection function set this variable to true in the next cycle
//When we have no connection to the backend then after Lynus_Standards.Constants_General.tTimeDissableLynusFunctions days the Function is dissabled with all of his functionalities
timResetConnectionOnGVL(IN:= NOT timResetConnectionOnGVL.Q, PT:= T#1H, Q=> , ET=> );
	IF timResetConnectionOnGVL.Q THEN Lynus_Standards.GVL_Communicator.bStateConnectionToEnableFunctions := FALSE; END_IF
		IF NOT Lynus_Standards.GVL_Communicator.bStateConnectionToEnableFunctions THEN timDissableFunctions.IN := TRUE; ELSE timDissableFunctions.IN := FALSE; END_IF  
			timDissableFunctions(IN:= , PT:= Lynus_Standards.Constants_General.tTimeDissableLynusFunctions, Q=> , ET=> );
	
(*------------------------------------------------------------------Error----------------------------------------------------------------------------*)	

IF timDissableFunctions.Q THEN fbEHE.bWarning := TRUE; fbEHE.iWarningCode := 0; ELSE fbEHE.bWarning := FALSE; END_IF 
	IF (Lynus_Standards.GVL_Energy.stNumberOfDevices.diNumberOfEHE > Constants_Energy.diMaxNumberOfElectricHeatingElements) OR 
		(Lynus_Standards.GVL_Sensors.stDataTemperatureSensors[diNrOfTempS_IN].bEnabled AND Lynus_Standards.GVL_Sensors.stDataTemperatureSensors[diNrOfTempS_IN].byErrorWarning = 2) OR
			fbGetSystemTime.ERR THEN 
				fbEHE.bError := TRUE; 
	ELSE 
				fbEHE.bError := FALSE; 
	END_IF

IF Lynus_Standards.GVL_Energy.stNumberOfDevices.diNumberOfEHE > Constants_Energy.diMaxNumberOfElectricHeatingElements THEN fbEHE.iErrorCode := 1;
ELSIF fbGetSystemTime.ERR THEN fbEHE.iErrorCode := 3;
ELSIF Lynus_Standards.GVL_Sensors.stDataTemperatureSensors[diNrOfTempS_IN].bEnabled AND Lynus_Standards.GVL_Sensors.stDataTemperatureSensors[diNrOfTempS_IN].byErrorWarning = 2 THEN fbEHE.iErrorCode := 2;
END_IF 

(*------------------------------------------------------------------Logic----------------------------------------------------------------------------*)
	
//Calcualte the total SOC if we have more then 1 battery in our system
diNumberOfActiveBatterys := 0;
	dwSumSOC := 0;
		FOR liLPBatteryData := 1 TO Constants_Energy.diMaxNumberOfBatterys BY 1 DO
			IF Lynus_Standards.GVL_Energy.stDataOfBatterys[diNrOfEMS_IN,liLPBatteryData].bEnabled THEN diNumberOfActiveBatterys := diNumberOfActiveBatterys + 1; END_IF
				dwSumSOC := dwSumSOC + Lynus_Standards.GVL_Energy.stDataOfBatterys[diNrOfEMS_IN,liLPBatteryData].dwSOC;
		END_FOR
	
IF diNumberOfActiveBatterys > 0 THEN
	fbEHE.dwBatterySOC := DINT_TO_DWORD(DWORD_TO_DINT(dwSumSOC) / diNumberOfActiveBatterys);
ELSE
	fbEHE.dwBatterySOC := 100;	//When we have no battery in the ems system
END_IF

//Check if one or more Batterysystems or batteryinverter make island mode
diNumberOfBatteryInverterInEPO := 0;
	FOR liLPInEPO := 1 TO Constants_Energy.diMaxNumberOfBatteryInverters BY 1 DO
		IF Lynus_Standards.GVL_Energy.stDataOfBatteryInverters[diNrOfEMS_IN,liLPInEPO].bWorkOnIslandMode THEN fbEHE.bEPOIsActive := TRUE; diNumberOfBatteryInverterInEPO := diNumberOfBatteryInverterInEPO + 1; END_IF
	END_FOR 
		IF diNumberOfBatteryInverterInEPO <= 0 THEN fbEHE.bEPOIsActive := FALSE; END_IF

//Check the max. power of the grid connection and the sum of grid power
lrSizeGridConnection := 0;
	lrGridPower := 0;
		FOR liLPGridData := 1 TO Constants_Energy.diMaxNumberOfGridConnections BY 1 DO
			lrSizeGridConnection := lrSizeGridConnection + Lynus_Standards.GVL_Energy.stDataGridConnections[diNrOfEMS_IN,liLPGridData].rSizeGridConn;
				lrGridPower := lrGridPower + Lynus_Standards.GVL_Energy.stDataGridConnections[diNrOfEMS_IN,liLPGridData].lrPower;
		END_FOR		
		
//Set the target power from the EMS to the EHE Function
fbEHE.arrTargetPower[1] := Lynus_Standards.GVL_Energy.stDataElectricHeatingElements[diNrOfEMS_IN,diNrOfEHE_OUT].arrTargetPowerEMS[1];

FOR byLPTargetPowerTo0 := 2 TO 10 BY 1 DO
	fbEHE.arrTargetPower[byLPTargetPowerTo0] := 0;
END_FOR
	stSetupEHE.rMaxPower2 := 0;
		stSetupEHE.rMaxPower3 := 0;
			stSetupEHE.rMaxPower4 := 0;
				stSetupEHE.rMaxPower5 := 0;
					stSetupEHE.rMaxPower6 := 0;
						stSetupEHE.rMaxPower7 := 0;
							stSetupEHE.rMaxPower8 := 0;
								stSetupEHE.rMaxPower9 := 0;
									stSetupEHE.rMaxPower10 := 0;

//Digital input for external lock signal
fbDIExternalLock(bInvers:= FALSE, bSignal=> );

//Functionblock EHE
fbEHE(
	bEnable:= bEnable AND NOT timDissableFunctions.Q,
	bError:= , 
	bIsStepSwitched:= FALSE, 
	bEPOIsActive:= , 
	bExternalLock:= fbDIExternalLock.bSignal, 
	bWriteWithDelay:= TRUE,
	bTimeDissableFunctions:= timDissableFunctions.Q,
	iErrorCode:= , 
	iWarningCode:= ,
	diNumberOfEHE:= diNrOfEHE_OUT, 
	dwBatterySOC:= , 
	lrSizeGridConnection:= lrSizeGridConnection,
	lrGridPower:= lrGridPower,
	lrTotalCounterEnergy_Consumption:= , 
	lrTotalCounterEnergy_Production:= , 
	lrCounterEnergyT1_Consumption:= , 
	lrCounterEnergyT2_Consumption:= , 
	lrCounterEnergyT1_Production:= , 
	lrCounterEnergyT2_Production:= , 
	lrPowerEHE:= , 
	arrTargetPower:= , 
	rTemperatureInBoiler:= Lynus_Standards.GVL_Sensors.stDataTemperatureSensors[diNrOfTempS_IN].rTemperature, 
	tTimDelayOutput:= T#5S, 
	stSystemTime:= , 
	stSetupEHE:= stSetupEHE, 
	stDataEHEOut=> , 
	stDataEHEOutDelay=> stDataEHE);
	
(*-------------------------------------------------------------------------Output----------------------------------------------------------------------*)

IF bNoLinear THEN 
	fbInterpolation.rXInputValue := (stSetupEHE.rMaxPower1 * fbEHE.stDataEHEOut.rTargetPower) / 100; 
		fbInterpolation.arrYIntermediateValues[1] := 10;
			fbInterpolation.arrYIntermediateValues[2] := 20;
				fbInterpolation.arrYIntermediateValues[3] := 30;
					fbInterpolation.arrYIntermediateValues[4] := 40;
						fbInterpolation.arrYIntermediateValues[5] := 50;
	fbInterpolation.arrYIntermediateValues[6] := 60;
		fbInterpolation.arrYIntermediateValues[7] := 70;
			fbInterpolation.arrYIntermediateValues[8] := 80;
				fbInterpolation.arrYIntermediateValues[9] := 90;
					fbInterpolation.arrYIntermediateValues[10] := 100;
	fbInterpolation(rXInputValue:=, arrXIntermediateValues:= arrTableOfInterpolationPoints, arrYIntermediateValues:=, rYOutputValue=> );
END_IF

IF bNoLinear THEN 
	fbAOEHE.rSignal := fbInterpolation.rYOutputValue;
	//Target Power, to use this on a external Function
	rTargetPowerForExtFunc := fbInterpolation.rYOutputValue;
ELSE
	fbAOEHE.rSignal := fbEHE.stDataEHEOut.rTargetPower;
	//Target Power, to use this on a external Function
	rTargetPowerForExtFunc := fbEHE.stDataEHEOut.rTargetPower;
END_IF

fbAOEHE(
	rYMinTerminalValue:= 0, 
	rXMinInputSignal:= 0, 
	rYMaxTerminalValue:= 32767, 
	rXMaxInputSignal:= 100, 
	rSignal:= , 
	usiState=> );

(*-----------------------------------------------------------Handle data to Global structure for the electric heating element-----------------------------------------------------------------*)

//Delte al old Data on GVL after a online change or change on the variable diNrOfEMS_IDOD
IF diNrOfEMS_IN <> diNrOfEMS_IN_CP AND iStateGVLData = 0 THEN iStateGVLData := 10; END_IF 

CASE iStateGVLData OF
	
	0://Init Step
		byWaitInStep := 0;
			diCounterForGVL := 1;
	
	1://Wait for 4 Steps before clean al Data on GVL
		byWaitInStep := byWaitInStep + 1;
			IF byWaitInStep >= 4 AND fbNumberDevice.bNumberIsCalculatet THEN iStateGVLData := 2; END_IF
				//To much Devices, back to the Init step
				IF byWaitInStep >= 4 AND NOT fbNumberDevice.bNumberIsCalculatet THEN iStateGVLData := 0; END_IF	
			
	2://Clear all Data in GVL
		FOR diLPForGVL := 1 TO Constants_Energy.diMaxNumberOfEMS BY 1 DO 
			Lynus_Standards.GVL_Energy.stDataElectricHeatingElements[diLPForGVL,diCounterForGVL].bEnabled := FALSE;
				Lynus_Standards.GVL_Energy.stDataElectricHeatingElements[diLPForGVL,diCounterForGVL].bIsStepSwitched := FALSE;
					Lynus_Standards.GVL_Energy.stDataElectricHeatingElements[diLPForGVL,diCounterForGVL].bIsControllable := FALSE;
						Lynus_Standards.GVL_Energy.stDataElectricHeatingElements[diLPForGVL,diCounterForGVL].byPriority := 0;
							Lynus_Standards.GVL_Energy.stDataElectricHeatingElements[diLPForGVL,diCounterForGVL].byErrorWarning := 0;
								Lynus_Standards.GVL_Energy.stDataElectricHeatingElements[diLPForGVL,diCounterForGVL].byNumberOfSteps := 0;
									Lynus_Standards.GVL_Energy.stDataElectricHeatingElements[diLPForGVL,diCounterForGVL].lrPower := 0;
										Lynus_Standards.GVL_Energy.stDataElectricHeatingElements[diLPForGVL,diCounterForGVL].lrPowerConsumption := 0;
											Lynus_Standards.GVL_Energy.stDataElectricHeatingElements[diLPForGVL,diCounterForGVL].lrPowerProduction := 0;
												FOR byLPGVLSetMaxPower := 1 TO 10 BY 1 DO
													Lynus_Standards.GVL_Energy.stDataElectricHeatingElements[diLPForGVL,diCounterForGVL].arrMaxPower[byLPGVLSetMaxPower] := 0;
												END_FOR 
													//Set also the target value from ems back here to 0 and not in EMS function because EMS is in Standy when we have a online change (Problem when we delete a ems function and make a online change)
													FOR byLPGVLSetMaxPower := 1 TO 10 BY 1 DO
														Lynus_Standards.GVL_Energy.stDataElectricHeatingElements[diLPForGVL,diCounterForGVL].arrTargetPowerEMS[byLPGVLSetMaxPower] := 0;	
													END_FOR
		END_FOR
			diCounterForGVL := diCounterForGVL + 1;
				diCounterForGVL := LIMIT(0,diCounterForGVL,Constants_Energy.diMaxNumberOfElectricHeatingElements);
					//Back to the init step
					IF diCounterForGVL >= Constants_Energy.diMaxNumberOfElectricHeatingElements THEN iStateGVLData := 0; END_IF

